Yaskawa INFORM job: DEMO_ROOF_SIDE_0625_3PAINT_6.JBI

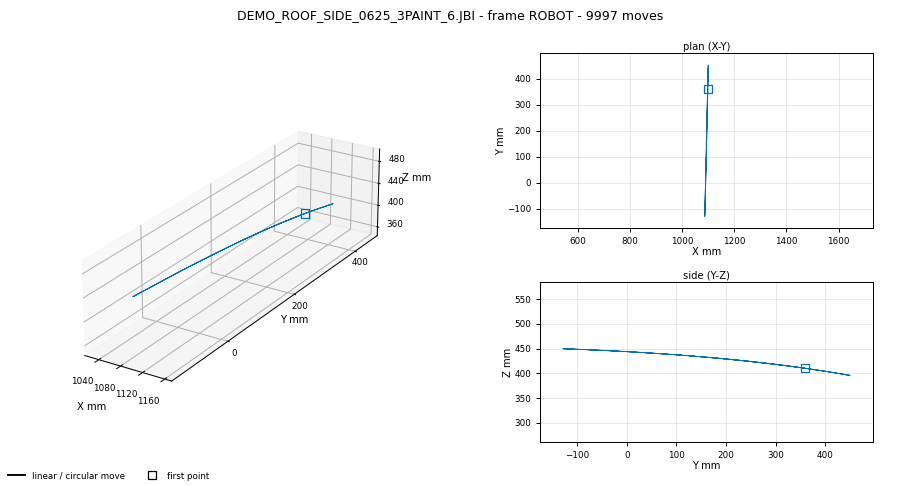
[picture p0: tool path of DEMO_ROOF_SIDE_0625_3PAINT_6.JBI in frame ROBOT, 9997 of 9997 moves have a stored position in this frame; points joined in program order, loops and branches not executed]
/JOB
//NAME DEMO_ROOF_SIDE_0625_3PAINT6
//POS
///NPOS 9997,0,0,0,0,0
///TOOL 0
///USER 0
///POSTYPE ROBOT
///RECTAN
///RCONF 1,0,0,0,0,0,0,0,0,0,0,0,0,0,0,0,0,0,0,0,0,0,0,0
C00000=1098.376,358.973,410.800,178.995,19.657,152.456
C00001=1098.369,358.726,410.835,178.993,19.653,152.456
C00002=1098.364,358.478,410.870,178.990,19.649,152.455
C00003=1098.358,358.230,410.905,178.986,19.645,152.455
C00004=1098.352,357.983,410.939,178.984,19.641,152.455
C00005=1098.347,357.735,410.974,178.980,19.637,152.454
C00006=1098.340,357.488,411.009,178.977,19.632,152.454
C00007=1098.332,357.110,411.062,178.973,19.626,152.453
C00008=1098.324,356.733,411.115,178.968,19.620,152.452
C00009=1098.314,356.355,411.168,178.964,19.614,152.452
C00010=1098.306,355.978,411.220,178.959,19.608,152.451
C00011=1098.300,355.731,411.256,178.956,19.604,152.451
C00012=1098.295,355.483,411.291,178.953,19.600,152.450
C00013=1098.289,355.235,411.325,178.950,19.596,152.450
C00014=1098.284,354.988,411.359,178.947,19.592,152.449
C00015=1098.277,354.740,411.395,178.944,19.588,152.449
C00016=1098.272,354.493,411.429,178.941,19.585,152.449
C00017=1098.266,354.245,411.463,178.938,19.580,152.448
C00018=1098.261,353.998,411.498,178.935,19.576,152.448
C00019=1098.254,353.750,411.532,178.932,19.572,152.447
C00020=1098.249,353.502,411.567,178.929,19.568,152.447
C00021=1098.243,353.255,411.601,178.926,19.565,152.446
C00022=1098.237,353.007,411.636,178.923,19.561,152.446
C00023=1098.231,352.760,411.671,178.919,19.557,152.446
C00024=1098.226,352.513,411.705,178.917,19.553,152.445
C00025=1098.220,352.265,411.740,178.913,19.549,152.445
C00026=1098.214,352.017,411.774,178.911,19.545,152.445
C00027=1098.208,351.770,411.808,178.907,19.541,152.444
C00028=1098.203,351.522,411.843,178.905,19.538,152.444
C00029=1098.197,351.275,411.877,178.901,19.534,152.443
C00030=1098.191,351.027,411.911,178.898,19.530,152.443
C00031=1098.186,350.779,411.945,178.895,19.526,152.443
C00032=1098.180,350.531,411.979,178.892,19.522,152.442
C00033=1098.174,350.284,412.013,178.889,19.519,152.442
C00034=1098.169,350.037,412.048,178.886,19.515,152.442
C00035=1098.163,349.789,412.082,178.883,19.512,152.441
C00036=1098.157,349.541,412.116,178.880,19.507,152.441
C00037=1098.151,349.294,412.150,178.877,19.504,152.441
C00038=1098.146,349.046,412.185,178.874,19.500,152.440
C00039=1098.140,348.799,412.218,178.871,19.497,152.440
C00040=1098.134,348.551,412.252,178.868,19.493,152.440
C00041=1098.128,348.303,412.287,178.865,19.489,152.439
C00042=1098.123,348.056,412.321,178.861,19.485,152.439
C00043=1098.117,347.808,412.355,178.859,19.482,152.439
C00044=1098.111,347.561,412.389,178.855,19.478,152.438
C00045=1098.105,347.313,412.423,178.853,19.475,152.438
C00046=1098.100,347.066,412.457,178.849,19.470,152.438
C00047=1098.095,346.818,412.491,178.847,19.467,152.437
C00048=1098.088,346.570,412.525,178.843,19.463,152.437
C00049=1098.082,346.322,412.559,178.840,19.460,152.437
C00050=1098.077,346.075,412.593,178.837,19.456,152.436
C00051=1098.071,345.827,412.627,178.834,19.453,152.436
C00052=1098.065,345.579,412.660,178.831,19.449,152.436
C00053=1098.060,345.332,412.695,178.828,19.445,152.435
C00054=1098.054,345.084,412.729,178.824,19.442,152.435
C00055=1098.049,344.837,412.762,178.822,19.438,152.435
C00056=1098.043,344.589,412.796,178.818,19.434,152.434
C00057=1098.038,344.341,412.830,178.815,19.431,152.434
C00058=1098.031,344.093,412.864,178.812,19.427,152.434
C00059=1098.022,343.718,412.915,178.808,19.422,152.433
C00060=1098.014,343.343,412.966,178.803,19.417,152.433
C00061=1098.005,342.968,413.017,178.798,19.412,152.433
C00062=1097.996,342.593,413.067,178.793,19.406,152.432
C00063=1097.990,342.345,413.101,178.790,19.403,152.432
C00064=1097.984,342.098,413.135,178.788,19.400,152.432
C00065=1097.979,341.850,413.169,178.784,19.396,152.431
C00066=1097.973,341.602,413.202,178.781,19.393,152.431
C00067=1097.967,341.354,413.236,178.778,19.389,152.431
C00068=1097.962,341.107,413.269,178.775,19.386,152.431
C00069=1097.956,340.859,413.303,178.771,19.382,152.430
C00070=1097.951,340.611,413.336,178.769,19.379,152.430
C00071=1097.945,340.363,413.370,178.766,19.376,152.430
C00072=1097.939,340.116,413.403,178.762,19.372,152.430
C00073=1097.934,339.868,413.437,178.759,19.369,152.429
C00074=1097.928,339.620,413.470,178.756,19.365,152.429
C00075=1097.922,339.373,413.503,178.753,19.362,152.429
C00076=1097.917,339.126,413.536,178.750,19.359,152.429
C00077=1097.911,338.878,413.570,178.747,19.355,152.428
C00078=1097.906,338.630,413.603,178.744,19.352,152.428
C00079=1097.900,338.382,413.636,178.740,19.349,152.428
C00080=1097.894,338.134,413.670,178.737,19.345,152.428
C00081=1097.888,337.887,413.703,178.735,19.342,152.427
C00082=1097.882,337.639,413.737,178.731,19.339,152.427
C00083=1097.877,337.391,413.770,178.728,19.335,152.427
C00084=1097.871,337.143,413.803,178.725,19.332,152.427
C00085=1097.865,336.896,413.836,178.722,19.329,152.427
C00086=1097.859,336.648,413.869,178.719,19.326,152.426
C00087=1097.854,336.400,413.903,178.715,19.322,152.426
C00088=1097.847,336.152,413.935,178.712,19.319,152.426
C00089=1097.842,335.904,413.969,178.709,19.316,152.426
C00090=1097.836,335.656,414.002,178.706,19.312,152.426
C00091=1097.831,335.409,414.035,178.703,19.309,152.425
C00092=1097.825,335.162,414.068,178.700,19.307,152.425
C00093=1097.820,334.914,414.101,178.696,19.303,152.425
C00094=1097.814,334.666,414.134,178.694,19.300,152.425
C00095=1097.808,334.418,414.167,178.691,19.297,152.424
C00096=1097.802,334.170,414.201,178.687,19.293,152.424
C00097=1097.797,333.922,414.233,178.684,19.290,152.424
C00098=1097.791,333.674,414.266,178.681,19.287,152.424
C00099=1097.786,333.427,414.299,178.678,19.283,152.424
C00100=1097.779,333.179,414.332,178.675,19.281,152.424
C00101=1097.774,332.932,414.365,178.672,19.278,152.423
C00102=1097.769,332.683,414.398,178.668,19.274,152.423
C00103=1097.762,332.435,414.430,178.665,19.271,152.423
C00104=1097.757,332.187,414.464,178.662,19.268,152.423
C00105=1097.751,331.941,414.496,178.659,19.265,152.423
C00106=1097.745,331.693,414.529,178.656,19.262,152.423
C00107=1097.739,331.444,414.561,178.653,19.259,152.422
C00108=1097.734,331.197,414.595,178.650,19.256,152.422
C00109=1097.728,330.949,414.627,178.646,19.253,152.422
C00110=1097.722,330.701,414.660,178.643,19.250,152.422
C00111=1097.713,330.320,414.710,178.638,19.245,152.422
C00112=1097.704,329.938,414.760,178.634,19.240,152.421
C00113=1097.695,329.558,414.811,178.628,19.236,152.421
C00114=1097.686,329.176,414.861,178.624,19.231,152.421
C00115=1097.680,328.929,414.893,178.620,19.228,152.421
C00116=1097.675,328.680,414.926,178.617,19.225,152.421
C00117=1097.669,328.432,414.959,178.614,19.222,152.421
C00118=1097.663,328.185,414.990,178.611,19.220,152.421
C00119=1097.658,327.937,415.024,178.607,19.216,152.420
C00120=1097.652,327.689,415.056,178.605,19.213,152.420
C00121=1097.645,327.441,415.088,178.602,19.211,152.420
C00122=1097.640,327.194,415.120,178.598,19.208,152.420
C00123=1097.634,326.946,415.153,178.595,19.204,152.420
C00124=1097.628,326.698,415.186,178.592,19.201,152.420
C00125=1097.622,326.450,415.218,178.589,19.199,152.420
C00126=1097.618,326.202,415.251,178.586,19.196,152.420
C00127=1097.612,325.954,415.283,178.582,19.193,152.420
C00128=1097.605,325.706,415.315,178.579,19.190,152.419
C00129=1097.600,325.459,415.347,178.576,19.187,152.419
C00130=1097.595,325.210,415.380,178.573,19.184,152.419
C00131=1097.588,324.963,415.412,178.569,19.181,152.419
C00132=1097.583,324.715,415.444,178.566,19.178,152.419
C00133=1097.577,324.467,415.476,178.563,19.175,152.419
C00134=1097.571,324.219,415.509,178.560,19.173,152.419
C00135=1097.566,323.972,415.541,178.557,19.170,152.419
C00136=1097.560,323.723,415.573,178.553,19.167,152.418
C00137=1097.554,323.475,415.605,178.550,19.164,152.418
C00138=1097.548,323.228,415.637,178.547,19.161,152.418
C00139=1097.543,322.980,415.670,178.544,19.158,152.418
C00140=1097.538,322.732,415.702,178.542,19.155,152.418
C00141=1097.532,322.484,415.734,178.538,19.152,152.418
C00142=1097.526,322.236,415.766,178.535,19.149,152.418
C00143=1097.520,321.989,415.798,178.532,19.147,152.418
C00144=1097.514,321.741,415.830,178.529,19.144,152.418
C00145=1097.509,321.493,415.862,178.526,19.141,152.418
C00146=1097.503,321.245,415.894,178.522,19.138,152.417
C00147=1097.497,320.996,415.926,178.519,19.135,152.417
C00148=1097.492,320.749,415.958,178.516,19.133,152.417
C00149=1097.486,320.501,415.990,178.513,19.130,152.417
C00150=1097.481,320.253,416.022,178.510,19.127,152.417
C00151=1097.475,320.005,416.054,178.507,19.125,152.417
C00152=1097.469,319.757,416.086,178.503,19.121,152.417
C00153=1097.464,319.509,416.118,178.500,19.119,152.417
C00154=1097.459,319.261,416.150,178.497,19.116,152.417
C00155=1097.453,319.013,416.182,178.494,19.113,152.417
C00156=1097.447,318.766,416.213,178.491,19.111,152.417
C00157=1097.441,318.517,416.246,178.488,19.108,152.417
C00158=1097.436,318.270,416.277,178.484,19.105,152.416
C00159=1097.430,318.022,416.309,178.481,19.102,152.416
C00160=1097.425,317.774,416.341,178.478,19.099,152.416
C00161=1097.419,317.527,416.373,178.475,19.097,152.416
C00162=1097.413,317.279,416.405,178.472,19.094,152.416
C00163=1097.405,316.890,416.454,178.466,19.089,152.416
C00164=1097.397,316.502,416.504,178.462,19.085,152.416
C00165=1097.387,316.114,416.553,178.456,19.081,152.416
C00166=1097.379,315.725,416.603,178.452,19.077,152.416
C00167=1097.373,315.478,416.635,178.449,19.074,152.416
C00168=1097.368,315.229,416.666,178.445,19.071,152.416
C00169=1097.362,314.981,416.698,178.442,19.068,152.416
C00170=1097.356,314.734,416.729,178.439,19.066,152.416
C00171=1097.350,314.486,416.761,178.435,19.063,152.416
C00172=1097.344,314.237,416.792,178.432,19.061,152.416
C00173=1097.338,313.990,416.823,178.429,19.058,152.416
C00174=1097.332,313.742,416.855,178.426,19.056,152.415
C00175=1097.327,313.494,416.886,178.423,19.053,152.416
C00176=1097.321,313.246,416.918,178.420,19.051,152.415
C00177=1097.315,312.998,416.949,178.416,19.047,152.415
C00178=1097.310,312.750,416.980,178.412,19.045,152.415
C00179=1097.303,312.502,417.012,178.409,19.043,152.415
C00180=1097.298,312.255,417.043,178.406,19.040,152.415
C00181=1097.292,312.006,417.075,178.403,19.038,152.415
C00182=1097.286,311.759,417.106,178.400,19.035,152.415
C00183=1097.280,311.510,417.137,178.397,19.033,152.415
C00184=1097.275,311.262,417.169,178.394,19.030,152.415
C00185=1097.269,311.014,417.199,178.391,19.028,152.415
C00186=1097.263,310.766,417.231,178.387,19.025,152.415
C00187=1097.257,310.518,417.261,178.384,19.023,152.415
C00188=1097.252,310.271,417.293,178.380,19.020,152.415
C00189=1097.246,310.022,417.324,178.377,19.017,152.415
C00190=1097.240,309.775,417.355,178.374,19.015,152.415
C00191=1097.235,309.527,417.386,178.371,19.013,152.415
C00192=1097.228,309.279,417.418,178.367,19.010,152.415
C00193=1097.223,309.031,417.449,178.364,19.008,152.415
C00194=1097.217,308.783,417.480,178.361,19.005,152.415
C00195=1097.212,308.535,417.511,178.358,19.003,152.415
C00196=1097.207,308.287,417.542,178.355,19.000,152.415
C00197=1097.200,308.039,417.573,178.352,18.998,152.415
C00198=1097.195,307.791,417.604,178.348,18.996,152.416
C00199=1097.189,307.543,417.635,178.345,18.993,152.415
C00200=1097.183,307.295,417.666,178.342,18.991,152.415
C00201=1097.178,307.047,417.697,178.339,18.988,152.415
C00202=1097.173,306.799,417.728,178.335,18.985,152.416
C00203=1097.166,306.551,417.758,178.332,18.983,152.416
C00204=1097.161,306.303,417.790,178.329,18.980,152.415
C00205=1097.155,306.055,417.820,178.325,18.978,152.416
C00206=1097.150,305.807,417.851,178.322,18.975,152.415
C00207=1097.143,305.559,417.882,178.319,18.973,152.416
C00208=1097.138,305.311,417.914,178.316,18.971,152.416
C00209=1097.132,305.063,417.944,178.313,18.968,152.416
C00210=1097.127,304.815,417.975,178.309,18.966,152.416
C00211=1097.121,304.567,418.005,178.306,18.963,152.416
C00212=1097.116,304.320,418.036,178.303,18.961,152.416
C00213=1097.110,304.071,418.067,178.300,18.958,152.416
C00214=1097.104,303.824,418.098,178.297,18.956,152.416
C00215=1097.096,303.437,418.145,178.291,18.952,152.416
C00216=1097.087,303.052,418.193,178.286,18.948,152.416
C00217=1097.077,302.666,418.241,178.281,18.945,152.416
C00218=1097.069,302.281,418.289,178.277,18.941,152.416
C00219=1097.064,302.032,418.320,178.273,18.939,152.416
C00220=1097.058,301.785,418.350,178.270,18.936,152.416
C00221=1097.052,301.537,418.381,178.267,18.934,152.416
C00222=1097.047,301.289,418.412,178.264,18.932,152.416
C00223=1097.041,301.041,418.442,178.260,18.928,152.416
C00224=1097.036,300.793,418.472,178.257,18.926,152.416
C00225=1097.031,300.545,418.503,178.253,18.924,152.416
C00226=1097.025,300.296,418.533,178.250,18.922,152.416
C00227=1097.019,300.049,418.563,178.247,18.919,152.416
C00228=1097.014,299.801,418.594,178.244,18.917,152.416
C00229=1097.008,299.553,418.624,178.240,18.914,152.416
C00230=1097.002,299.305,418.655,178.237,18.912,152.416
C00231=1096.997,299.057,418.686,178.234,18.910,152.416
C00232=1096.992,298.809,418.716,178.231,18.907,152.416
C00233=1096.986,298.560,418.746,178.228,18.905,152.416
C00234=1096.981,298.312,418.777,178.224,18.903,152.416
C00235=1096.975,298.065,418.807,178.221,18.900,152.417
C00236=1096.969,297.816,418.838,178.218,18.898,152.417
C00237=1096.963,297.568,418.867,178.214,18.896,152.417
C00238=1096.957,297.320,418.898,178.211,18.894,152.417
C00239=1096.952,297.072,418.928,178.208,18.891,152.417
C00240=1096.947,296.824,418.959,178.205,18.889,152.417
C00241=1096.941,296.575,418.989,178.202,18.887,152.417
C00242=1096.935,296.328,419.019,178.199,18.885,152.417
C00243=1096.929,296.080,419.049,178.196,18.883,152.417
C00244=1096.924,295.831,419.079,178.193,18.880,152.417
C00245=1096.918,295.583,419.109,178.189,18.878,152.417
C00246=1096.912,295.336,419.140,178.186,18.876,152.417
C00247=1096.907,295.087,419.169,178.183,18.874,152.417
C00248=1096.901,294.839,419.200,178.179,18.871,152.417
C00249=1096.895,294.591,419.229,178.176,18.869,152.418
C00250=1096.890,294.343,419.260,178.173,18.867,152.418
C00251=1096.884,294.095,419.289,178.169,18.865,152.418
C00252=1096.878,293.847,419.320,178.166,18.863,152.418
C00253=1096.872,293.599,419.350,178.163,18.860,152.418
C00254=1096.867,293.351,419.380,178.160,18.858,152.418
C00255=1096.861,293.103,419.410,178.156,18.856,152.418
C00256=1096.856,292.854,419.440,178.153,18.854,152.418
C00257=1096.850,292.606,419.469,178.150,18.851,152.418
C00258=1096.844,292.358,419.500,178.146,18.849,152.418
C00259=1096.839,292.110,419.529,178.143,18.847,152.418
C00260=1096.833,291.862,419.560,178.140,18.845,152.418
C00261=1096.828,291.614,419.589,178.137,18.842,152.419
C00262=1096.822,291.366,419.619,178.134,18.841,152.419
C00263=1096.816,291.118,419.648,178.131,18.839,152.419
C00264=1096.810,290.870,419.678,178.127,18.837,152.419
C00265=1096.805,290.622,419.708,178.124,18.834,152.419
C00266=1096.799,290.373,419.738,178.121,18.832,152.419
C00267=1096.791,290.001,419.783,178.116,18.829,152.419
C00268=1096.782,289.630,419.827,178.111,18.826,152.419
C00269=1096.774,289.258,419.872,178.106,18.822,152.420
C00270=1096.765,288.887,419.916,178.101,18.819,152.420
C00271=1096.759,288.638,419.946,178.098,18.817,152.420
C00272=1096.754,288.390,419.975,178.095,18.815,152.420
C00273=1096.748,288.141,420.005,178.092,18.813,152.420
C00274=1096.742,287.894,420.035,178.088,18.811,152.420
C00275=1096.736,287.645,420.064,178.085,18.809,152.420
C00276=1096.731,287.398,420.094,178.082,18.807,152.420
C00277=1096.726,287.149,420.123,178.078,18.805,152.420
C00278=1096.720,286.901,420.152,178.075,18.802,152.421
C00279=1096.714,286.653,420.182,178.071,18.801,152.421
C00280=1096.709,286.404,420.211,178.068,18.798,152.421
C00281=1096.702,286.157,420.241,178.066,18.797,152.421
C00282=1096.697,285.909,420.270,178.062,18.794,152.421
C00283=1096.692,285.660,420.300,178.059,18.793,152.421
C00284=1096.685,285.412,420.329,178.056,18.790,152.421
C00285=1096.680,285.164,420.359,178.052,18.788,152.421
C00286=1096.674,284.915,420.388,178.049,18.786,152.422
C00287=1096.669,284.668,420.417,178.046,18.784,152.422
C00288=1096.663,284.420,420.447,178.042,18.782,152.422
C00289=1096.658,284.171,420.476,178.040,18.780,152.422
C00290=1096.651,283.923,420.505,178.036,18.778,152.422
C00291=1096.646,283.675,420.535,178.033,18.776,152.422
C00292=1096.641,283.427,420.564,178.030,18.774,152.422
C00293=1096.635,283.179,420.593,178.026,18.772,152.422
C00294=1096.629,282.930,420.623,178.023,18.770,152.423
C00295=1096.624,282.681,420.652,178.020,18.767,152.423
C00296=1096.618,282.434,420.681,178.016,18.766,152.423
C00297=1096.613,282.185,420.710,178.014,18.764,152.423
C00298=1096.607,281.937,420.739,178.010,18.762,152.423
C00299=1096.602,281.689,420.769,178.007,18.760,152.423
C00300=1096.595,281.441,420.798,178.004,18.758,152.423
C00301=1096.590,281.193,420.827,178.000,18.755,152.423
C00302=1096.584,280.944,420.856,177.997,18.754,152.424
C00303=1096.579,280.696,420.885,177.994,18.751,152.424
C00304=1096.573,280.448,420.914,177.991,18.750,152.424
C00305=1096.567,280.200,420.943,177.988,18.748,152.424
C00306=1096.561,279.951,420.972,177.984,18.746,152.424
C00307=1096.556,279.703,421.001,177.981,18.744,152.424
C00308=1096.550,279.455,421.030,177.977,18.741,152.424
C00309=1096.545,279.207,421.060,177.974,18.740,152.425
C00310=1096.539,278.959,421.088,177.971,18.738,152.425
C00311=1096.533,278.711,421.117,177.968,18.736,152.425
C00312=1096.528,278.462,421.146,177.965,18.734,152.425
C00313=1096.522,278.214,421.174,177.961,18.732,152.425
C00314=1096.517,277.966,421.204,177.958,18.730,152.425
C00315=1096.511,277.717,421.232,177.954,18.728,152.426
C00316=1096.505,277.469,421.261,177.952,18.726,152.426
C00317=1096.500,277.221,421.291,177.948,18.724,152.426
C00318=1096.494,276.972,421.319,177.945,18.722,152.426
C00319=1096.486,276.610,421.361,177.940,18.719,152.426
C00320=1096.478,276.248,421.403,177.936,18.717,152.427
C00321=1096.469,275.885,421.445,177.931,18.714,152.427
C00322=1096.460,275.523,421.487,177.926,18.711,152.427
C00323=1096.456,275.275,421.515,177.923,18.709,152.427
C00324=1096.450,275.026,421.545,177.920,18.707,152.427
C00325=1096.444,274.778,421.573,177.916,18.705,152.427
C00326=1096.439,274.530,421.602,177.913,18.703,152.428
C00327=1096.433,274.281,421.630,177.910,18.702,152.428
C00328=1096.427,274.034,421.659,177.907,18.700,152.428
C00329=1096.421,273.785,421.687,177.903,18.698,152.428
C00330=1096.416,273.536,421.716,177.900,18.696,152.428
C00331=1096.410,273.289,421.745,177.896,18.694,152.428
C00332=1096.404,273.040,421.773,177.894,18.692,152.429
C00333=1096.399,272.792,421.802,177.890,18.690,152.429
C00334=1096.393,272.544,421.830,177.887,18.688,152.429
C00335=1096.388,272.295,421.859,177.884,18.686,152.429
C00336=1096.382,272.046,421.887,177.881,18.685,152.429
C00337=1096.376,271.798,421.916,177.877,18.683,152.430
C00338=1096.371,271.550,421.944,177.874,18.681,152.430
C00339=1096.365,271.302,421.973,177.871,18.679,152.430
C00340=1096.359,271.054,422.001,177.867,18.677,152.430
C00341=1096.353,270.805,422.030,177.865,18.676,152.430
C00342=1096.349,270.557,422.058,177.861,18.674,152.430
C00343=1096.343,270.308,422.086,177.858,18.671,152.430
C00344=1096.337,270.060,422.114,177.854,18.670,152.431
C00345=1096.331,269.812,422.143,177.852,18.668,152.431
C00346=1096.326,269.564,422.171,177.848,18.666,152.431
C00347=1096.320,269.315,422.200,177.845,18.664,152.431
C00348=1096.314,269.067,422.228,177.841,18.663,152.431
C00349=1096.308,268.818,422.256,177.838,18.660,152.432
C00350=1096.303,268.570,422.284,177.835,18.659,152.432
C00351=1096.297,268.322,422.312,177.832,18.657,152.432
C00352=1096.292,268.074,422.341,177.828,18.655,152.432
C00353=1096.286,267.825,422.369,177.825,18.653,152.432
C00354=1096.280,267.577,422.397,177.822,18.652,152.433
C00355=1096.274,267.329,422.426,177.819,18.650,152.433
C00356=1096.269,267.081,422.454,177.815,18.648,152.433
C00357=1096.263,266.832,422.482,177.812,18.646,152.433
C00358=1096.258,266.584,422.510,177.809,18.644,152.433
C00359=1096.252,266.335,422.538,177.806,18.643,152.433
C00360=1096.246,266.087,422.566,177.802,18.641,152.434
C00361=1096.241,265.839,422.594,177.799,18.639,152.434
C00362=1096.235,265.590,422.622,177.796,18.637,152.434
C00363=1096.230,265.342,422.650,177.793,18.636,152.434
C00364=1096.224,265.093,422.678,177.789,18.634,152.434
C00365=1096.219,264.845,422.706,177.786,18.631,152.435
C00366=1096.213,264.597,422.734,177.783,18.630,152.435
C00367=1096.207,264.348,422.762,177.780,18.628,152.435
C00368=1096.201,264.100,422.790,177.776,18.627,152.435
C00369=1096.195,263.851,422.818,177.773,18.625,152.435
C00370=1096.190,263.603,422.846,177.770,18.623,152.436
C00371=1096.182,263.243,422.885,177.765,18.621,152.436
C00372=1096.173,262.884,422.926,177.760,18.618,152.436
C00373=1096.165,262.525,422.966,177.756,18.616,152.437
C00374=1096.157,262.164,423.006,177.751,18.613,152.437
C00375=1096.151,261.916,423.034,177.748,18.612,152.437
C00376=1096.145,261.668,423.062,177.745,18.610,152.437
C00377=1096.139,261.420,423.090,177.741,18.608,152.438
C00378=1096.134,261.171,423.117,177.738,18.606,152.438
C00379=1096.128,260.923,423.145,177.735,18.605,152.438
C00380=1096.122,260.674,423.173,177.731,18.603,152.438
C00381=1096.116,260.426,423.201,177.728,18.602,152.439
C00382=1096.111,260.178,423.228,177.725,18.600,152.439
C00383=1096.105,259.929,423.256,177.722,18.598,152.439
C00384=1096.100,259.680,423.283,177.718,18.596,152.439
C00385=1096.094,259.432,423.311,177.716,18.595,152.439
C00386=1096.088,259.184,423.339,177.712,18.593,152.440
C00387=1096.083,258.935,423.366,177.709,18.591,152.440
C00388=1096.076,258.687,423.394,177.705,18.590,152.440
C00389=1096.071,258.438,423.421,177.702,18.588,152.440
C00390=1096.065,258.190,423.449,177.699,18.586,152.440
C00391=1096.060,257.942,423.476,177.695,18.584,152.441
C00392=1096.054,257.693,423.504,177.693,18.583,152.441
C00393=1096.048,257.445,423.531,177.689,18.581,152.441
C00394=1096.043,257.196,423.559,177.686,18.580,152.441
C00395=1096.037,256.948,423.585,177.683,18.578,152.442
C00396=1096.031,256.699,423.614,177.679,18.576,152.442
C00397=1096.026,256.451,423.641,177.676,18.575,152.442
C00398=1096.020,256.203,423.668,177.673,18.573,152.442
C00399=1096.015,255.954,423.695,177.670,18.571,152.442
C00400=1096.008,255.706,423.723,177.666,18.569,152.443
C00401=1096.003,255.457,423.750,177.664,18.568,152.443
C00402=1095.997,255.209,423.777,177.660,18.566,152.443
C00403=1095.992,254.961,423.805,177.657,18.565,152.443
C00404=1095.986,254.712,423.832,177.654,18.563,152.444
C00405=1095.980,254.464,423.860,177.650,18.562,152.444
C00406=1095.974,254.215,423.887,177.647,18.560,152.444
C00407=1095.969,253.966,423.914,177.644,18.558,152.444
C00408=1095.963,253.719,423.941,177.641,18.556,152.444
C00409=1095.958,253.469,423.969,177.637,18.554,152.445
C00410=1095.952,253.221,423.996,177.635,18.553,152.445
C00411=1095.947,252.972,424.023,177.631,18.551,152.445
C00412=1095.941,252.725,424.050,177.628,18.550,152.445
C00413=1095.936,252.476,424.077,177.625,18.548,152.446
C00414=1095.930,252.228,424.104,177.621,18.547,152.446
C00415=1095.924,251.978,424.132,177.618,18.544,152.446
C00416=1095.919,251.730,424.158,177.615,18.543,152.446
C00417=1095.913,251.482,424.186,177.612,18.541,152.446
C00418=1095.908,251.233,424.213,177.608,18.540,152.447
C00419=1095.902,250.985,424.240,177.606,18.538,152.447
C00420=1095.897,250.736,424.267,177.602,18.536,152.447
C00421=1095.892,250.488,424.294,177.598,18.535,152.447
C00422=1095.886,250.239,424.321,177.596,18.533,152.448
C00423=1095.877,249.877,424.361,177.591,18.531,152.448
C00424=1095.869,249.514,424.400,177.586,18.528,152.448
C00425=1095.862,249.152,424.439,177.582,18.526,152.448
C00426=1095.853,248.789,424.479,177.576,18.523,152.449
C00427=1095.847,248.540,424.506,177.574,18.522,152.449
C00428=1095.842,248.292,424.532,177.570,18.520,152.449
C00429=1095.837,248.043,424.559,177.567,18.518,152.449
C00430=1095.831,247.795,424.586,177.564,18.517,152.450
C00431=1095.826,247.546,424.613,177.561,18.515,152.450
C00432=1095.820,247.298,424.640,177.558,18.514,152.450
C00433=1095.814,247.050,424.667,177.554,18.512,152.450
C00434=1095.809,246.801,424.693,177.551,18.510,152.451
C00435=1095.804,246.553,424.721,177.548,18.509,152.451
C00436=1095.798,246.304,424.747,177.545,18.507,152.451
C00437=1095.792,246.055,424.773,177.541,18.505,152.451
C00438=1095.786,245.807,424.800,177.538,18.504,152.452
C00439=1095.781,245.559,424.826,177.535,18.502,152.452
C00440=1095.776,245.310,424.854,177.532,18.501,152.452
C00441=1095.770,245.062,424.880,177.529,18.499,152.452
C00442=1095.764,244.813,424.907,177.525,18.498,152.453
C00443=1095.758,244.565,424.934,177.522,18.496,152.453
C00444=1095.753,244.316,424.960,177.519,18.495,152.453
C00445=1095.748,244.067,424.987,177.516,18.493,152.453
C00446=1095.742,243.819,425.013,177.513,18.492,152.454
C00447=1095.736,243.570,425.040,177.509,18.490,152.454
C00448=1095.731,243.321,425.066,177.506,18.489,152.454
C00449=1095.725,243.073,425.093,177.503,18.487,152.454
C00450=1095.719,242.825,425.119,177.500,18.486,152.454
C00451=1095.714,242.576,425.146,177.497,18.484,152.455
C00452=1095.708,242.327,425.172,177.493,18.482,152.455
C00453=1095.702,242.079,425.199,177.490,18.481,152.455
C00454=1095.697,241.831,425.225,177.487,18.479,152.455
C00455=1095.691,241.582,425.251,177.484,18.478,152.456
C00456=1095.685,241.333,425.278,177.481,18.476,152.456
C00457=1095.679,241.085,425.304,177.478,18.475,152.456
C00458=1095.674,240.836,425.330,177.474,18.473,152.456
C00459=1095.668,240.588,425.357,177.471,18.471,152.457
C00460=1095.663,240.339,425.383,177.468,18.470,152.457
C00461=1095.657,240.090,425.410,177.465,18.468,152.457
C00462=1095.651,239.842,425.436,177.462,18.467,152.457
C00463=1095.646,239.593,425.462,177.458,18.466,152.458
C00464=1095.640,239.345,425.489,177.454,18.464,152.458
C00465=1095.635,239.096,425.515,177.452,18.462,152.458
C00466=1095.629,238.847,425.541,177.448,18.461,152.459
C00467=1095.623,238.598,425.567,177.446,18.459,152.459
C00468=1095.618,238.350,425.594,177.442,18.458,152.459
C00469=1095.613,238.102,425.620,177.439,18.456,152.459
C00470=1095.607,237.853,425.646,177.436,18.455,152.460
C00471=1095.601,237.604,425.672,177.433,18.453,152.460
C00472=1095.595,237.356,425.698,177.429,18.452,152.460
C00473=1095.589,237.107,425.724,177.426,18.450,152.460
C00474=1095.584,236.858,425.750,177.423,18.449,152.460
C00475=1095.576,236.489,425.789,177.419,18.447,152.461
C00476=1095.567,236.120,425.827,177.413,18.444,152.461
C00477=1095.559,235.751,425.867,177.409,18.442,152.462
C00478=1095.551,235.381,425.905,177.404,18.440,152.462
C00479=1095.545,235.133,425.931,177.401,18.438,152.462
C00480=1095.540,234.884,425.957,177.398,18.437,152.463
C00481=1095.534,234.635,425.983,177.394,18.435,152.463
C00482=1095.529,234.386,426.009,177.392,18.434,152.463
C00483=1095.523,234.138,426.035,177.388,18.432,152.463
C00484=1095.517,233.889,426.061,177.385,18.431,152.464
C00485=1095.512,233.640,426.087,177.382,18.429,152.464
C00486=1095.506,233.392,426.113,177.378,18.427,152.464
C00487=1095.500,233.143,426.139,177.375,18.427,152.464
C00488=1095.495,232.895,426.164,177.372,18.425,152.465
C00489=1095.489,232.646,426.190,177.369,18.424,152.465
C00490=1095.484,232.397,426.216,177.366,18.422,152.465
C00491=1095.478,232.149,426.242,177.363,18.421,152.465
C00492=1095.472,231.900,426.268,177.359,18.419,152.466
C00493=1095.467,231.652,426.294,177.357,18.418,152.466
C00494=1095.461,231.403,426.319,177.353,18.416,152.466
C00495=1095.456,231.154,426.345,177.350,18.415,152.466
C00496=1095.450,230.905,426.371,177.347,18.413,152.467
C00497=1095.445,230.657,426.397,177.344,18.412,152.467
C00498=1095.439,230.408,426.422,177.340,18.410,152.467
C00499=1095.433,230.159,426.448,177.338,18.409,152.468
C00500=1095.427,229.911,426.474,177.334,18.407,152.468
C00501=1095.422,229.663,426.499,177.331,18.406,152.468
C00502=1095.416,229.414,426.525,177.328,18.404,152.468
C00503=1095.410,229.165,426.551,177.325,18.404,152.469
C00504=1095.404,228.917,426.576,177.321,18.402,152.469
C00505=1095.399,228.668,426.602,177.319,18.401,152.469
C00506=1095.394,228.419,426.628,177.315,18.399,152.469
C00507=1095.388,228.171,426.653,177.312,18.398,152.470
C00508=1095.382,227.922,426.679,177.309,18.396,152.470
C00509=1095.377,227.674,426.704,177.306,18.395,152.470
C00510=1095.371,227.425,426.730,177.302,18.393,152.471
C00511=1095.365,227.176,426.754,177.300,18.392,152.471
C00512=1095.360,226.927,426.780,177.296,18.390,152.471
C00513=1095.354,226.679,426.805,177.293,18.389,152.471
C00514=1095.349,226.430,426.831,177.290,18.387,152.472
C00515=1095.343,226.182,426.856,177.287,18.386,152.472
C00516=1095.337,225.933,426.881,177.283,18.385,152.472
C00517=1095.331,225.684,426.907,177.281,18.383,152.472
C00518=1095.326,225.436,426.932,177.277,18.382,152.473
C00519=1095.321,225.186,426.958,177.274,18.380,152.473
C00520=1095.314,224.938,426.983,177.271,18.379,152.473
C00521=1095.310,224.689,427.009,177.268,18.378,152.474
C00522=1095.303,224.441,427.034,177.264,18.376,152.474
C00523=1095.298,224.192,427.060,177.262,18.375,152.474
C00524=1095.293,223.943,427.084,177.258,18.373,152.474
C00525=1095.286,223.695,427.109,177.255,18.372,152.475
C00526=1095.282,223.446,427.135,177.252,18.370,152.475
C00527=1095.273,223.068,427.174,177.247,18.368,152.475
C00528=1095.265,222.689,427.211,177.243,18.366,152.476
C00529=1095.256,222.312,427.250,177.238,18.364,152.476
C00530=1095.247,221.934,427.288,177.233,18.362,152.477
C00531=1095.242,221.685,427.314,177.230,18.360,152.477
C00532=1095.236,221.436,427.338,177.227,18.360,152.477
C00533=1095.230,221.188,427.363,177.224,18.358,152.477
C00534=1095.225,220.940,427.388,177.221,18.357,152.478
C00535=1095.219,220.690,427.414,177.217,18.355,152.478
C00536=1095.213,220.442,427.439,177.214,18.354,152.478
C00537=1095.208,220.193,427.463,177.211,18.352,152.479
C00538=1095.202,219.944,427.488,177.208,18.351,152.479
C00539=1095.197,219.695,427.513,177.205,18.349,152.479
C00540=1095.191,219.447,427.539,177.202,18.348,152.479
C00541=1095.186,219.198,427.563,177.198,18.347,152.480
C00542=1095.179,218.949,427.588,177.195,18.345,152.480
C00543=1095.174,218.701,427.612,177.193,18.344,152.480
C00544=1095.169,218.452,427.638,177.189,18.342,152.480
C00545=1095.163,218.203,427.663,177.186,18.342,152.481
C00546=1095.157,217.955,427.688,177.183,18.340,152.481
C00547=1095.151,217.705,427.713,177.180,18.339,152.481
C00548=1095.146,217.457,427.738,177.176,18.337,152.482
C00549=1095.140,217.208,427.762,177.174,18.336,152.482
C00550=1095.135,216.960,427.788,177.171,18.335,152.482
C00551=1095.130,216.711,427.812,177.167,18.333,152.483
C00552=1095.124,216.462,427.837,177.164,18.332,152.483
C00553=1095.118,216.214,427.862,177.161,18.330,152.483
C00554=1095.112,215.965,427.886,177.158,18.329,152.483
C00555=1095.107,215.717,427.911,177.154,18.328,152.484
C00556=1095.101,215.467,427.936,177.152,18.326,152.484
C00557=1095.095,215.219,427.960,177.149,18.325,152.484
C00558=1095.090,214.970,427.986,177.145,18.323,152.484
C00559=1095.085,214.721,428.010,177.143,18.322,152.485
C00560=1095.079,214.473,428.035,177.139,18.321,152.485
C00561=1095.073,214.223,428.059,177.136,18.320,152.485
C00562=1095.068,213.975,428.084,177.133,18.319,152.486
C00563=1095.062,213.726,428.109,177.130,18.317,152.486
C00564=1095.057,213.478,428.133,177.127,18.316,152.486
C00565=1095.051,213.229,428.157,177.124,18.314,152.486
C00566=1095.045,212.980,428.183,177.121,18.313,152.487
C00567=1095.040,212.732,428.207,177.118,18.312,152.487
C00568=1095.034,212.482,428.232,177.114,18.310,152.487
C00569=1095.029,212.234,428.256,177.112,18.309,152.487
C00570=1095.023,211.985,428.280,177.108,18.307,152.488
C00571=1095.017,211.737,428.305,177.105,18.306,152.488
C00572=1095.012,211.488,428.330,177.102,18.305,152.488
C00573=1095.006,211.239,428.354,177.099,18.303,152.489
C00574=1095.001,210.990,428.378,177.096,18.302,152.489
C00575=1094.995,210.742,428.403,177.092,18.301,152.489
C00576=1094.989,210.492,428.427,177.090,18.300,152.490
C00577=1094.984,210.244,428.452,177.087,18.298,152.490
C00578=1094.978,209.995,428.475,177.083,18.297,152.490
C00579=1094.970,209.621,428.512,177.079,18.295,152.490
C00580=1094.961,209.247,428.549,177.074,18.293,152.491
C00581=1094.952,208.872,428.585,177.070,18.291,152.491
C00582=1094.944,208.498,428.622,177.065,18.289,152.492
C00583=1094.921,207.483,428.720,177.011,18.266,152.497
C00584=1094.916,207.234,428.744,177.008,18.266,152.497
C00585=1094.910,206.986,428.768,177.005,18.265,152.498
C00586=1094.904,206.737,428.793,177.002,18.265,152.498
C00587=1094.899,206.488,428.816,176.998,18.264,152.499
C00588=1094.893,206.239,428.840,176.995,18.264,152.499
C00589=1094.888,205.991,428.864,176.991,18.263,152.500
C00590=1094.882,205.741,428.889,176.988,18.262,152.500
C00591=1094.876,205.492,428.912,176.985,18.262,152.501
C00592=1094.871,205.244,428.936,176.982,18.262,152.501
C00593=1094.865,204.996,428.960,176.979,18.261,152.502
C00594=1094.860,204.746,428.983,176.975,18.261,152.502
C00595=1094.855,204.498,429.007,176.972,18.261,152.503
C00596=1094.848,204.249,429.031,176.969,18.260,152.503
C00597=1094.843,204.000,429.055,176.966,18.260,152.504
C00598=1094.837,203.751,429.079,176.963,18.259,152.504
C00599=1094.832,203.503,429.103,176.960,18.259,152.505
C00600=1094.827,203.254,429.126,176.956,18.258,152.505
C00601=1094.821,203.005,429.150,176.953,18.258,152.506
C00602=1094.816,202.756,429.174,176.949,18.257,152.506
C00603=1094.809,202.507,429.198,176.946,18.256,152.507
C00604=1094.804,202.258,429.221,176.943,18.256,152.507
C00605=1094.798,202.010,429.245,176.940,18.256,152.508
C00606=1094.792,201.761,429.268,176.937,18.255,152.508
C00607=1094.787,201.512,429.292,176.933,18.255,152.509
C00608=1094.780,201.263,429.316,176.930,18.255,152.509
C00609=1094.775,201.014,429.340,176.927,18.254,152.510
C00610=1094.769,200.766,429.363,176.924,18.254,152.510
C00611=1094.764,200.517,429.386,176.921,18.253,152.511
C00612=1094.758,200.268,429.410,176.917,18.253,152.511
C00613=1094.752,200.019,429.433,176.914,18.253,152.512
C00614=1094.747,199.770,429.456,176.911,18.252,152.512
C00615=1094.741,199.521,429.481,176.908,18.252,152.513
C00616=1094.735,199.272,429.504,176.905,18.251,152.514
C00617=1094.729,199.024,429.528,176.902,18.251,152.514
C00618=1094.724,198.775,429.551,176.898,18.250,152.514
C00619=1094.718,198.526,429.574,176.895,18.250,152.515
C00620=1094.712,198.278,429.598,176.892,18.249,152.515
C00621=1094.707,198.028,429.621,176.889,18.249,152.516
C00622=1094.701,197.780,429.645,176.886,18.249,152.517
C00623=1094.696,197.531,429.668,176.882,18.248,152.517
C00624=1094.691,197.282,429.691,176.879,18.247,152.517
C00625=1094.685,197.034,429.715,176.875,18.247,152.518
C00626=1094.678,196.784,429.738,176.872,18.246,152.518
C00627=1094.673,196.535,429.762,176.869,18.246,152.519
C00628=1094.667,196.286,429.785,176.866,18.245,152.519
C00629=1094.661,196.038,429.809,176.863,18.245,152.520
C00630=1094.656,195.788,429.832,176.860,18.245,152.520
C00631=1094.651,195.540,429.855,176.857,18.244,152.521
C00632=1094.645,195.291,429.878,176.853,18.244,152.521
C00633=1094.639,195.042,429.902,176.851,18.243,152.522
C00634=1094.634,194.793,429.925,176.847,18.243,152.522
C00635=1094.628,194.544,429.948,176.844,18.243,152.523
C00636=1094.622,194.295,429.971,176.841,18.242,152.523
C00637=1094.617,194.047,429.994,176.838,18.242,152.524
C00638=1094.611,193.798,430.018,176.835,18.241,152.524
C00639=1094.606,193.549,430.041,176.832,18.241,152.525
C00640=1094.600,193.300,430.064,176.829,18.240,152.525
C00641=1094.594,193.051,430.087,176.825,18.240,152.526
C00642=1094.589,192.802,430.111,176.822,18.239,152.526
C00643=1094.584,192.553,430.134,176.819,18.239,152.527
C00644=1094.577,192.278,430.159,176.816,18.238,152.527
C00645=1094.572,192.003,430.184,176.812,18.237,152.528
C00646=1094.565,191.729,430.210,176.809,18.237,152.528
C00647=1094.559,191.453,430.235,176.806,18.237,152.529
C00648=1094.553,191.204,430.258,176.803,18.236,152.529
C00649=1094.548,190.955,430.281,176.799,18.236,152.530
C00650=1094.543,190.706,430.305,176.796,18.235,152.530
C00651=1094.537,190.457,430.328,176.793,18.235,152.531
C00652=1094.531,190.208,430.351,176.790,18.234,152.531
C00653=1094.526,189.959,430.374,176.787,18.234,152.532
C00654=1094.520,189.710,430.397,176.784,18.233,152.532
C00655=1094.515,189.462,430.419,176.781,18.233,152.533
C00656=1094.510,189.213,430.443,176.778,18.232,152.533
C00657=1094.504,188.964,430.466,176.774,18.232,152.534
C00658=1094.498,188.715,430.489,176.771,18.231,152.534
C00659=1094.493,188.466,430.512,176.768,18.230,152.534
C00660=1094.487,188.217,430.535,176.765,18.230,152.535
C00661=1094.481,187.968,430.557,176.762,18.229,152.535
C00662=1094.476,187.720,430.580,176.759,18.229,152.536
C00663=1094.471,187.471,430.604,176.756,18.228,152.536
C00664=1094.465,187.222,430.627,176.753,18.228,152.537
C00665=1094.460,186.973,430.649,176.750,18.227,152.537
C00666=1094.454,186.724,430.672,176.747,18.227,152.538
C00667=1094.449,186.476,430.694,176.744,18.226,152.538
C00668=1094.443,186.227,430.717,176.740,18.226,152.539
C00669=1094.437,185.978,430.740,176.737,18.225,152.539
C00670=1094.432,185.729,430.763,176.734,18.224,152.539
C00671=1094.426,185.479,430.785,176.731,18.224,152.540
C00672=1094.421,185.231,430.808,176.728,18.223,152.540
C00673=1094.415,184.982,430.831,176.725,18.223,152.541
C00674=1094.410,184.733,430.854,176.722,18.222,152.541
C00675=1094.404,184.484,430.876,176.719,18.222,152.542
C00676=1094.399,184.235,430.899,176.716,18.221,152.542
C00677=1094.392,183.986,430.921,176.713,18.221,152.543
C00678=1094.386,183.737,430.944,176.710,18.220,152.543
C00679=1094.381,183.488,430.967,176.706,18.220,152.544
C00680=1094.375,183.239,430.990,176.703,18.219,152.544
C00681=1094.370,182.991,431.012,176.700,18.219,152.545
C00682=1094.364,182.742,431.034,176.697,18.218,152.545
C00683=1094.358,182.493,431.057,176.694,18.218,152.545
C00684=1094.352,182.244,431.080,176.692,18.218,152.546
C00685=1094.347,181.995,431.103,176.689,18.217,152.546
C00686=1094.341,181.746,431.124,176.685,18.217,152.547
C00687=1094.335,181.498,431.147,176.682,18.216,152.547
C00688=1094.330,181.248,431.169,176.679,18.216,152.548
C00689=1094.324,180.999,431.192,176.676,18.215,152.548
C00690=1094.318,180.751,431.214,176.673,18.215,152.549
C00691=1094.312,180.501,431.237,176.670,18.214,152.549
C00692=1094.307,180.252,431.259,176.667,18.213,152.550
C00693=1094.301,180.004,431.281,176.664,18.213,152.550
C00694=1094.295,179.755,431.304,176.661,18.213,152.551
C00695=1094.290,179.505,431.326,176.657,18.212,152.551
C00696=1094.283,179.257,431.348,176.654,18.212,152.552
C00697=1094.278,179.008,431.371,176.651,18.211,152.552
C00698=1094.273,178.759,431.393,176.648,18.211,152.553
C00699=1094.267,178.510,431.416,176.645,18.210,152.553
C00700=1094.261,178.261,431.438,176.642,18.209,152.553
C00701=1094.256,178.012,431.460,176.640,18.209,152.554
C00702=1094.250,177.763,431.482,176.637,18.209,152.554
C00703=1094.244,177.514,431.504,176.634,18.208,152.555
C00704=1094.239,177.265,431.527,176.631,18.208,152.555
C00705=1094.233,177.017,431.548,176.628,18.207,152.556
C00706=1094.227,176.768,431.571,176.625,18.206,152.556
C00707=1094.222,176.518,431.593,176.621,18.206,152.557
C00708=1094.215,176.243,431.618,176.618,18.205,152.557
C00709=1094.210,175.967,431.642,176.615,18.205,152.558
C00710=1094.203,175.692,431.667,176.611,18.204,152.558
C00711=1094.197,175.416,431.691,176.608,18.204,152.559
C00712=1094.191,175.167,431.714,176.605,18.203,152.559
C00713=1094.185,174.918,431.736,176.602,18.202,152.559
C00714=1094.181,174.669,431.758,176.599,18.202,152.560
C00715=1094.174,174.421,431.780,176.596,18.201,152.560
C00716=1094.169,174.172,431.802,176.593,18.201,152.561
C00717=1094.163,173.922,431.824,176.591,18.200,152.561
C00718=1094.157,173.674,431.847,176.588,18.200,152.562
C00719=1094.153,173.425,431.868,176.585,18.199,152.562
C00720=1094.146,173.176,431.890,176.581,18.199,152.562
C00721=1094.141,172.926,431.912,176.578,18.198,152.563
C00722=1094.135,172.678,431.934,176.575,18.197,152.563
C00723=1094.130,172.429,431.957,176.572,18.197,152.564
C00724=1094.124,172.179,431.978,176.569,18.196,152.564
C00725=1094.119,171.931,432.000,176.566,18.195,152.565
C00726=1094.112,171.682,432.022,176.563,18.195,152.565
C00727=1094.107,171.433,432.044,176.561,18.195,152.565
C00728=1094.102,171.184,432.066,176.558,18.194,152.566
C00729=1094.096,170.935,432.088,176.555,18.193,152.566
C00730=1094.091,170.686,432.110,176.552,18.193,152.567
C00731=1094.085,170.436,432.132,176.549,18.192,152.567
C00732=1094.080,170.188,432.153,176.546,18.191,152.567
C00733=1094.074,169.939,432.176,176.543,18.191,152.568
C00734=1094.069,169.690,432.198,176.540,18.190,152.568
C00735=1094.063,169.441,432.219,176.537,18.190,152.569
C00736=1094.058,169.192,432.241,176.534,18.189,152.569
C00737=1094.052,168.943,432.263,176.532,18.189,152.570
C00738=1094.047,168.694,432.285,176.529,18.188,152.570
C00739=1094.041,168.445,432.306,176.526,18.187,152.570
C00740=1094.036,168.196,432.328,176.523,18.187,152.571
C00741=1094.030,167.947,432.350,176.520,18.186,152.571
C00742=1094.025,167.698,432.372,176.517,18.185,152.572
C00743=1094.019,167.449,432.393,176.514,18.184,152.572
C00744=1094.014,167.200,432.415,176.511,18.184,152.572
C00745=1094.008,166.951,432.437,176.508,18.183,152.573
C00746=1094.003,166.702,432.459,176.506,18.183,152.573
C00747=1093.997,166.453,432.480,176.503,18.182,152.574
C00748=1093.992,166.204,432.502,176.500,18.181,152.574
C00749=1093.986,165.955,432.524,176.497,18.181,152.574
C00750=1093.980,165.706,432.545,176.494,18.180,152.575
C00751=1093.975,165.457,432.567,176.491,18.179,152.575
C00752=1093.969,165.208,432.589,176.488,18.179,152.576
C00753=1093.964,164.959,432.611,176.485,18.178,152.576
C00754=1093.958,164.710,432.632,176.482,18.178,152.577
C00755=1093.953,164.462,432.654,176.480,18.177,152.577
C00756=1093.947,164.212,432.675,176.477,18.176,152.577
C00757=1093.942,163.963,432.696,176.474,18.175,152.578
C00758=1093.936,163.714,432.718,176.471,18.174,152.578
C00759=1093.931,163.465,432.740,176.468,18.174,152.578
C00760=1093.926,163.216,432.761,176.465,18.173,152.579
C00761=1093.920,162.967,432.783,176.462,18.172,152.579
C00762=1093.915,162.718,432.804,176.460,18.172,152.580
C00763=1093.909,162.469,432.826,176.457,18.172,152.580
C00764=1093.904,162.220,432.847,176.454,18.171,152.580
C00765=1093.899,161.971,432.869,176.451,18.170,152.581
C00766=1093.893,161.721,432.890,176.448,18.169,152.581
C00767=1093.887,161.473,432.911,176.445,18.168,152.581
C00768=1093.881,161.224,432.933,176.442,18.168,152.582
C00769=1093.876,160.975,432.954,176.440,18.167,152.582
C00770=1093.871,160.726,432.975,176.437,18.167,152.583
C00771=1093.865,160.477,432.997,176.434,18.166,152.583
C00772=1093.858,160.201,433.021,176.431,18.165,152.584
C00773=1093.853,159.926,433.044,176.428,18.165,152.584
C00774=1093.846,159.649,433.067,176.424,18.164,152.585
C00775=1093.840,159.373,433.091,176.421,18.163,152.585
C00776=1093.834,159.125,433.113,176.418,18.162,152.585
C00777=1093.828,158.875,433.134,176.416,18.162,152.586
C00778=1093.823,158.626,433.155,176.413,18.161,152.586
C00779=1093.817,158.378,433.176,176.410,18.160,152.586
C00780=1093.811,158.128,433.197,176.407,18.160,152.587
C00781=1093.807,157.879,433.219,176.404,18.159,152.587
C00782=1093.801,157.629,433.240,176.401,18.158,152.588
C00783=1093.795,157.381,433.261,176.399,18.158,152.588
C00784=1093.790,157.132,433.282,176.396,18.157,152.588
C00785=1093.784,156.883,433.303,176.393,18.157,152.589
C00786=1093.778,156.634,433.325,176.390,18.156,152.589
C00787=1093.773,156.385,433.345,176.387,18.155,152.589
C00788=1093.767,156.136,433.367,176.384,18.154,152.590
C00789=1093.762,155.887,433.387,176.382,18.154,152.590
C00790=1093.756,155.638,433.409,176.379,18.153,152.591
C00791=1093.750,155.388,433.429,176.376,18.153,152.591
C00792=1093.745,155.140,433.451,176.373,18.151,152.591
C00793=1093.739,154.891,433.471,176.370,18.151,152.592
C00794=1093.733,154.641,433.493,176.367,18.150,152.592
C00795=1093.728,154.392,433.514,176.365,18.150,152.593
C00796=1093.722,154.144,433.535,176.362,18.149,152.593
C00797=1093.717,153.894,433.556,176.359,18.148,152.593
C00798=1093.711,153.645,433.577,176.356,18.147,152.594
C00799=1093.706,153.396,433.598,176.353,18.147,152.594
C00800=1093.700,153.147,433.619,176.351,18.146,152.594
C00801=1093.694,152.898,433.640,176.348,18.146,152.595
C00802=1093.689,152.649,433.660,176.345,18.145,152.595
C00803=1093.683,152.400,433.682,176.342,18.144,152.596
C00804=1093.678,152.151,433.702,176.339,18.143,152.596
C00805=1093.672,151.901,433.723,176.336,18.142,152.596
C00806=1093.667,151.653,433.744,176.334,18.142,152.597
C00807=1093.661,151.403,433.765,176.331,18.141,152.597
C00808=1093.655,151.155,433.786,176.328,18.140,152.597
C00809=1093.649,150.906,433.806,176.325,18.140,152.598
C00810=1093.644,150.657,433.827,176.323,18.139,152.598
C00811=1093.638,150.407,433.848,176.321,18.138,152.598
C00812=1093.633,150.158,433.869,176.318,18.138,152.599
C00813=1093.627,149.909,433.890,176.315,18.137,152.599
C00814=1093.622,149.660,433.910,176.312,18.136,152.600
C00815=1093.617,149.412,433.932,176.309,18.135,152.600
C00816=1093.610,149.162,433.952,176.307,18.135,152.600
C00817=1093.605,148.913,433.972,176.304,18.134,152.601
C00818=1093.600,148.664,433.993,176.301,18.133,152.601
C00819=1093.594,148.415,434.014,176.298,18.132,152.601
C00820=1093.588,148.166,434.035,176.295,18.131,152.602
C00821=1093.582,147.917,434.055,176.293,18.131,152.602
C00822=1093.577,147.668,434.076,176.290,18.130,152.602
C00823=1093.572,147.418,434.096,176.287,18.129,152.603
C00824=1093.565,147.169,434.118,176.284,18.129,152.603
C00825=1093.559,146.920,434.138,176.281,18.128,152.604
C00826=1093.554,146.671,434.158,176.279,18.127,152.604
C00827=1093.549,146.422,434.179,176.276,18.127,152.604
C00828=1093.543,146.173,434.199,176.273,18.126,152.605
C00829=1093.537,145.924,434.220,176.271,18.125,152.605
C00830=1093.532,145.674,434.240,176.269,18.125,152.605
C00831=1093.526,145.426,434.262,176.266,18.124,152.606
C00832=1093.520,145.177,434.282,176.263,18.123,152.606
C00833=1093.515,144.928,434.302,176.260,18.122,152.606
C00834=1093.510,144.679,434.323,176.257,18.121,152.607
C00835=1093.503,144.429,434.343,176.255,18.121,152.607
C00836=1093.497,144.154,434.366,176.252,18.120,152.607
C00837=1093.491,143.877,434.388,176.249,18.119,152.608
C00838=1093.486,143.601,434.411,176.245,18.118,152.608
C00839=1093.479,143.325,434.434,176.242,18.117,152.609
C00840=1093.473,143.076,434.454,176.240,18.117,152.609
C00841=1093.468,142.827,434.474,176.238,18.116,152.609
C00842=1093.463,142.577,434.495,176.235,18.115,152.610
C00843=1093.457,142.329,434.515,176.232,18.114,152.610
C00844=1093.451,142.079,434.536,176.229,18.113,152.610
C00845=1093.445,141.830,434.556,176.227,18.112,152.611
C00846=1093.440,141.581,434.576,176.224,18.112,152.611
C00847=1093.434,141.332,434.597,176.221,18.111,152.611
C00848=1093.428,141.083,434.617,176.218,18.110,152.612
C00849=1093.423,140.834,434.637,176.216,18.109,152.612
C00850=1093.418,140.585,434.658,176.213,18.109,152.612
C00851=1093.412,140.336,434.678,176.211,18.107,152.613
C00852=1093.407,140.087,434.698,176.208,18.107,152.613
C00853=1093.401,139.837,434.718,176.206,18.106,152.613
C00854=1093.396,139.588,434.738,176.203,18.105,152.614
C00855=1093.389,139.339,434.758,176.200,18.104,152.614
C00856=1093.384,139.090,434.779,176.197,18.104,152.614
C00857=1093.378,138.841,434.799,176.195,18.103,152.614
C00858=1093.372,138.592,434.819,176.192,18.102,152.615
C00859=1093.366,138.343,434.839,176.189,18.101,152.615
C00860=1093.362,138.093,434.859,176.186,18.100,152.616
C00861=1093.356,137.844,434.879,176.184,18.100,152.616
C00862=1093.350,137.595,434.900,176.181,18.099,152.616
C00863=1093.344,137.346,434.920,176.179,18.098,152.617
C00864=1093.339,137.097,434.940,176.176,18.097,152.617
C00865=1093.333,136.848,434.960,176.174,18.097,152.617
C00866=1093.327,136.599,434.979,176.171,18.095,152.617
C00867=1093.322,136.350,435.000,176.168,18.095,152.618
C00868=1093.316,136.101,435.020,176.165,18.094,152.618
C00869=1093.311,135.851,435.040,176.163,18.093,152.618
C00870=1093.305,135.602,435.060,176.160,18.092,152.619
C00871=1093.299,135.354,435.080,176.158,18.091,152.619
C00872=1093.294,135.104,435.100,176.155,18.090,152.619
C00873=1093.288,134.855,435.120,176.153,18.090,152.620
C00874=1093.283,134.606,435.140,176.150,18.089,152.620
C00875=1093.277,134.357,435.159,176.147,18.088,152.620
C00876=1093.271,134.108,435.179,176.144,18.087,152.621
C00877=1093.266,133.859,435.200,176.142,18.087,152.621
C00878=1093.260,133.609,435.219,176.139,18.086,152.621
C00879=1093.255,133.360,435.240,176.137,18.084,152.622
C00880=1093.249,133.111,435.260,176.134,18.084,152.622
C00881=1093.243,132.862,435.279,176.132,18.083,152.622
C00882=1093.238,132.613,435.299,176.129,18.082,152.622
C00883=1093.232,132.363,435.319,176.126,18.081,152.623
C00884=1093.226,132.114,435.339,176.124,18.081,152.623
C00885=1093.221,131.865,435.358,176.121,18.079,152.623
C00886=1093.216,131.616,435.378,176.118,18.079,152.624
C00887=1093.210,131.367,435.398,176.116,18.078,152.624
C00888=1093.204,131.118,435.418,176.114,18.077,152.624
C00889=1093.198,130.869,435.438,176.111,18.076,152.625
C00890=1093.192,130.619,435.457,176.108,18.075,152.625
C00891=1093.187,130.370,435.477,176.106,18.075,152.625
C00892=1093.181,130.121,435.497,176.103,18.074,152.626
C00893=1093.175,129.872,435.517,176.100,18.073,152.626
C00894=1093.170,129.623,435.536,176.097,18.072,152.626
C00895=1093.164,129.374,435.556,176.095,18.071,152.627
C00896=1093.158,129.124,435.575,176.093,18.070,152.627
C00897=1093.153,128.875,435.596,176.090,18.069,152.627
C00898=1093.147,128.626,435.615,176.088,18.069,152.627
C00899=1093.141,128.376,435.634,176.085,18.068,152.628
C00900=1093.134,128.101,435.656,176.082,18.067,152.628
C00901=1093.128,127.824,435.678,176.079,18.066,152.628
C00902=1093.122,127.548,435.699,176.077,18.065,152.629
C00903=1093.116,127.272,435.721,176.074,18.064,152.629
C00904=1093.110,127.022,435.740,176.071,18.063,152.629
C00905=1093.104,126.774,435.760,176.068,18.062,152.630
C00906=1093.099,126.524,435.780,176.066,18.061,152.630
C00907=1093.093,126.275,435.799,176.063,18.060,152.630
C00908=1093.087,126.026,435.819,176.060,18.059,152.631
C00909=1093.081,125.777,435.838,176.059,18.059,152.631
C00910=1093.076,125.527,435.858,176.056,18.057,152.631
C00911=1093.071,125.279,435.877,176.053,18.056,152.631
C00912=1093.065,125.029,435.897,176.051,18.056,152.632
C00913=1093.060,124.780,435.916,176.048,18.055,152.632
C00914=1093.054,124.531,435.936,176.045,18.054,152.632
C00915=1093.048,124.282,435.955,176.043,18.053,152.633
C00916=1093.042,124.032,435.974,176.041,18.052,152.633
C00917=1093.037,123.783,435.994,176.038,18.051,152.633
C00918=1093.031,123.535,436.013,176.035,18.050,152.633
C00919=1093.026,123.285,436.032,176.033,18.050,152.634
C00920=1093.020,123.036,436.052,176.030,18.048,152.634
C00921=1093.014,122.786,436.071,176.028,18.047,152.634
C00922=1093.008,122.538,436.091,176.026,18.047,152.634
C00923=1093.003,122.289,436.110,176.023,18.046,152.635
C00924=1092.997,122.039,436.129,176.020,18.044,152.635
C00925=1092.992,121.790,436.148,176.018,18.044,152.635
C00926=1092.986,121.540,436.168,176.016,18.043,152.636
C00927=1092.980,121.291,436.187,176.013,18.041,152.636
C00928=1092.975,121.043,436.206,176.010,18.040,152.636
C00929=1092.969,120.794,436.226,176.008,18.040,152.636
C00930=1092.964,120.544,436.245,176.006,18.039,152.637
C00931=1092.958,120.295,436.264,176.003,18.038,152.637
C00932=1092.953,120.046,436.283,176.001,18.037,152.637
C00933=1092.947,119.796,436.302,175.998,18.036,152.637
C00934=1092.941,119.547,436.321,175.995,18.035,152.638
C00935=1092.936,119.298,436.341,175.993,18.034,152.638
C00936=1092.931,119.049,436.360,175.991,18.033,152.638
C00937=1092.925,118.799,436.379,175.988,18.032,152.639
C00938=1092.919,118.550,436.398,175.986,18.031,152.639
C00939=1092.914,118.301,436.417,175.983,18.030,152.639
C00940=1092.908,118.052,436.437,175.981,18.029,152.639
C00941=1092.903,117.803,436.456,175.979,18.028,152.639
C00942=1092.897,117.554,436.475,175.976,18.027,152.640
C00943=1092.892,117.305,436.494,175.973,18.026,152.640
C00944=1092.886,117.055,436.514,175.971,18.025,152.640
C00945=1092.880,116.806,436.533,175.969,18.024,152.640
C00946=1092.876,116.557,436.551,175.966,18.023,152.641
C00947=1092.870,116.307,436.570,175.964,18.022,152.641
C00948=1092.864,116.058,436.589,175.961,18.021,152.641
C00949=1092.859,115.809,436.608,175.959,18.020,152.641
C00950=1092.853,115.560,436.628,175.957,18.019,152.642
C00951=1092.848,115.310,436.647,175.954,18.018,152.642
C00952=1092.843,115.061,436.666,175.951,18.016,152.642
C00953=1092.836,114.812,436.684,175.950,18.016,152.642
C00954=1092.831,114.563,436.704,175.947,18.015,152.643
C00955=1092.825,114.314,436.722,175.944,18.013,152.643
C00956=1092.820,114.065,436.742,175.942,18.013,152.643
C00957=1092.814,113.815,436.761,175.939,18.012,152.643
C00958=1092.808,113.566,436.779,175.937,18.010,152.644
C00959=1092.803,113.317,436.798,175.935,18.010,152.644
C00960=1092.797,113.067,436.817,175.932,18.009,152.644
C00961=1092.792,112.818,436.836,175.929,18.008,152.644
C00962=1092.786,112.570,436.854,175.928,18.006,152.645
C00963=1092.780,112.320,436.874,175.925,18.005,152.645
C00964=1092.774,112.044,436.894,175.922,18.004,152.645
C00965=1092.768,111.767,436.915,175.919,18.003,152.645
C00966=1092.761,111.491,436.936,175.917,18.002,152.646
C00967=1092.755,111.215,436.956,175.914,18.001,152.646
C00968=1092.750,110.965,436.976,175.912,18.000,152.646
C00969=1092.744,110.717,436.994,175.909,17.999,152.646
C00970=1092.738,110.467,437.013,175.907,17.998,152.647
C00971=1092.733,110.217,437.032,175.905,17.997,152.647
C00972=1092.727,109.969,437.050,175.902,17.996,152.647
C00973=1092.721,109.719,437.069,175.899,17.995,152.647
C00974=1092.716,109.470,437.088,175.898,17.994,152.648
C00975=1092.710,109.221,437.106,175.895,17.993,152.648
C00976=1092.704,108.971,437.125,175.893,17.992,152.648
C00977=1092.698,108.723,437.144,175.890,17.991,152.648
C00978=1092.693,108.473,437.162,175.887,17.990,152.649
C00979=1092.687,108.224,437.181,175.886,17.989,152.649
C00980=1092.682,107.975,437.200,175.883,17.987,152.649
C00981=1092.676,107.725,437.218,175.880,17.986,152.649
C00982=1092.670,107.477,437.236,175.878,17.986,152.649
C00983=1092.665,107.227,437.256,175.876,17.984,152.650
C00984=1092.659,106.977,437.274,175.873,17.983,152.650
C00985=1092.654,106.729,437.292,175.871,17.982,152.650
C00986=1092.648,106.479,437.311,175.869,17.981,152.650
C00987=1092.642,106.230,437.329,175.867,17.980,152.651
C00988=1092.637,105.981,437.349,175.864,17.979,152.651
C00989=1092.630,105.731,437.366,175.861,17.978,152.651
C00990=1092.625,105.482,437.385,175.860,17.977,152.651
C00991=1092.619,105.233,437.403,175.857,17.976,152.652
C00992=1092.614,104.984,437.422,175.854,17.974,152.652
C00993=1092.608,104.734,437.440,175.852,17.974,152.652
C00994=1092.603,104.485,437.459,175.850,17.972,152.652
C00995=1092.597,104.236,437.477,175.848,17.972,152.652
C00996=1092.592,103.987,437.496,175.845,17.970,152.653
C00997=1092.586,103.737,437.514,175.843,17.969,152.653
C00998=1092.581,103.488,437.533,175.841,17.968,152.653
C00999=1092.574,103.239,437.550,175.838,17.967,152.653
C01000=1092.569,102.990,437.569,175.835,17.966,152.653
C01001=1092.563,102.740,437.587,175.834,17.965,152.654
C01002=1092.558,102.492,437.606,175.831,17.963,152.654
C01003=1092.552,102.242,437.624,175.829,17.963,152.654
C01004=1092.547,101.992,437.642,175.827,17.961,152.654
C01005=1092.541,101.743,437.661,175.824,17.960,152.654
C01006=1092.536,101.494,437.679,175.822,17.959,152.655
C01007=1092.530,101.245,437.698,175.820,17.958,152.655
C01008=1092.525,100.995,437.716,175.817,17.957,152.655
C01009=1092.518,100.746,437.735,175.815,17.956,152.655
C01010=1092.513,100.497,437.752,175.812,17.954,152.655
C01011=1092.508,100.247,437.771,175.811,17.954,152.656
C01012=1092.502,99.999,437.789,175.808,17.953,152.656
C01013=1092.496,99.749,437.807,175.805,17.951,152.656
C01014=1092.491,99.500,437.825,175.803,17.950,152.656
C01015=1092.484,99.251,437.844,175.801,17.949,152.657
C01016=1092.479,99.002,437.861,175.799,17.948,152.657
C01017=1092.473,98.752,437.880,175.796,17.947,152.657
C01018=1092.468,98.503,437.898,175.794,17.946,152.657
C01019=1092.462,98.253,437.916,175.792,17.945,152.657
C01020=1092.457,98.004,437.934,175.789,17.944,152.658
C01021=1092.451,97.754,437.952,175.788,17.942,152.658
C01022=1092.445,97.506,437.970,175.785,17.941,152.658
C01023=1092.439,97.257,437.988,175.782,17.940,152.658
C01024=1092.434,97.007,438.006,175.780,17.939,152.658
C01025=1092.428,96.758,438.024,175.778,17.938,152.659
C01026=1092.422,96.509,438.043,175.776,17.937,152.659
C01027=1092.416,96.260,438.060,175.773,17.936,152.659
C01028=1092.410,95.983,438.081,175.771,17.934,152.659
C01029=1092.404,95.707,438.101,175.768,17.933,152.659
C01030=1092.398,95.431,438.121,175.765,17.932,152.660
C01031=1092.391,95.154,438.140,175.764,17.931,152.660
C01032=1092.386,94.905,438.159,175.761,17.929,152.660
C01033=1092.380,94.656,438.177,175.759,17.928,152.660
C01034=1092.375,94.407,438.194,175.757,17.927,152.660
C01035=1092.369,94.158,438.212,175.754,17.926,152.661
C01036=1092.364,93.907,438.230,175.752,17.925,152.661
C01037=1092.358,93.658,438.248,175.750,17.923,152.661
C01038=1092.352,93.409,438.266,175.747,17.922,152.661
C01039=1092.346,93.160,438.284,175.745,17.921,152.661
C01040=1092.341,92.911,438.302,175.743,17.919,152.661
C01041=1092.335,92.661,438.320,175.741,17.919,152.662
C01042=1092.330,92.412,438.338,175.739,17.917,152.662
C01043=1092.324,92.163,438.355,175.737,17.917,152.662
C01044=1092.318,91.913,438.373,175.734,17.915,152.662
C01045=1092.313,91.664,438.391,175.731,17.914,152.662
C01046=1092.308,91.415,438.409,175.730,17.913,152.662
C01047=1092.302,91.165,438.427,175.727,17.911,152.663
C01048=1092.296,90.916,438.445,175.725,17.910,152.663
C01049=1092.291,90.667,438.462,175.723,17.909,152.663
C01050=1092.285,90.417,438.480,175.721,17.908,152.663
C01051=1092.279,90.168,438.498,175.719,17.907,152.663
C01052=1092.274,89.919,438.515,175.716,17.905,152.664
C01053=1092.268,89.670,438.533,175.714,17.904,152.664
C01054=1092.262,89.421,438.551,175.711,17.903,152.664
C01055=1092.256,89.171,438.569,175.710,17.902,152.664
C01056=1092.250,88.922,438.586,175.707,17.901,152.664
C01057=1092.245,88.673,438.604,175.705,17.900,152.664
C01058=1092.239,88.423,438.622,175.703,17.899,152.665
C01059=1092.233,88.174,438.639,175.700,17.897,152.665
C01060=1092.228,87.925,438.657,175.699,17.896,152.665
C01061=1092.222,87.675,438.675,175.696,17.895,152.665
C01062=1092.216,87.426,438.692,175.694,17.894,152.665
C01063=1092.211,87.176,438.709,175.691,17.893,152.666
C01064=1092.205,86.927,438.727,175.690,17.891,152.666
C01065=1092.199,86.678,438.745,175.687,17.890,152.666
C01066=1092.194,86.429,438.762,175.685,17.889,152.666
C01067=1092.188,86.180,438.780,175.683,17.888,152.666
C01068=1092.182,85.930,438.798,175.681,17.886,152.666
C01069=1092.177,85.681,438.815,175.679,17.885,152.667
C01070=1092.171,85.431,438.832,175.676,17.884,152.667
C01071=1092.166,85.182,438.850,175.674,17.883,152.667
C01072=1092.160,84.932,438.868,175.672,17.881,152.667
C01073=1092.154,84.683,438.885,175.670,17.880,152.667
C01074=1092.149,84.434,438.903,175.668,17.879,152.667
C01075=1092.144,84.185,438.920,175.665,17.878,152.668
C01076=1092.137,83.935,438.937,175.663,17.876,152.668
C01077=1092.131,83.686,438.955,175.661,17.875,152.668
C01078=1092.126,83.437,438.972,175.659,17.874,152.668
C01079=1092.120,83.188,438.990,175.656,17.873,152.668
C01080=1092.114,82.938,439.007,175.655,17.871,152.668
C01081=1092.109,82.689,439.024,175.652,17.870,152.668
C01082=1092.103,82.440,439.042,175.650,17.869,152.669
C01083=1092.098,82.190,439.059,175.648,17.868,152.669
C01084=1092.093,81.941,439.076,175.646,17.866,152.669
C01085=1092.086,81.691,439.094,175.644,17.865,152.669
C01086=1092.081,81.442,439.112,175.641,17.864,152.669
C01087=1092.075,81.193,439.128,175.639,17.863,152.669
C01088=1092.069,80.944,439.146,175.637,17.861,152.669
C01089=1092.064,80.695,439.163,175.635,17.860,152.670
C01090=1092.058,80.444,439.181,175.633,17.859,152.670
C01091=1092.053,80.195,439.198,175.631,17.858,152.670
C01092=1092.047,79.919,439.217,175.628,17.856,152.670
C01093=1092.041,79.643,439.236,175.626,17.854,152.670
C01094=1092.034,79.367,439.256,175.624,17.853,152.670
C01095=1092.028,79.091,439.274,175.621,17.852,152.671
C01096=1092.022,78.842,439.292,175.619,17.850,152.671
C01097=1092.017,78.592,439.309,175.617,17.849,152.671
C01098=1092.011,78.343,439.326,175.615,17.848,152.671
C01099=1092.005,78.093,439.343,175.613,17.846,152.671
C01100=1092.000,77.844,439.361,175.611,17.845,152.671
C01101=1091.994,77.594,439.377,175.608,17.844,152.671
C01102=1091.988,77.345,439.394,175.607,17.843,152.671
C01103=1091.983,77.096,439.412,175.604,17.841,152.672
C01104=1091.977,76.847,439.429,175.602,17.841,152.672
C01105=1091.971,76.597,439.446,175.600,17.839,152.672
C01106=1091.965,76.348,439.463,175.598,17.838,152.672
C01107=1091.960,76.099,439.481,175.596,17.836,152.672
C01108=1091.954,75.849,439.497,175.594,17.835,152.672
C01109=1091.948,75.600,439.514,175.591,17.833,152.672
C01110=1091.943,75.351,439.531,175.590,17.833,152.673
C01111=1091.937,75.102,439.548,175.587,17.831,152.673
C01112=1091.931,74.851,439.565,175.585,17.830,152.673
C01113=1091.926,74.602,439.582,175.583,17.828,152.673
C01114=1091.920,74.353,439.599,175.581,17.827,152.673
C01115=1091.914,74.103,439.616,175.579,17.826,152.673
C01116=1091.909,73.854,439.634,175.576,17.824,152.673
C01117=1091.903,73.605,439.650,175.574,17.823,152.674
C01118=1091.897,73.356,439.668,175.572,17.822,152.674
C01119=1091.892,73.106,439.684,175.570,17.821,152.674
C01120=1091.886,72.857,439.701,175.568,17.819,152.674
C01121=1091.881,72.608,439.718,175.566,17.818,152.674
C01122=1091.875,72.359,439.734,175.564,17.816,152.674
C01123=1091.869,72.109,439.752,175.562,17.815,152.674
C01124=1091.863,71.859,439.769,175.560,17.814,152.674
C01125=1091.857,71.610,439.785,175.558,17.813,152.675
C01126=1091.852,71.361,439.803,175.556,17.811,152.675
C01127=1091.846,71.111,439.819,175.554,17.810,152.675
C01128=1091.841,70.862,439.836,175.551,17.809,152.675
C01129=1091.835,70.613,439.854,175.550,17.808,152.675
C01130=1091.829,70.363,439.870,175.547,17.806,152.675
C01131=1091.824,70.114,439.887,175.545,17.805,152.675
C01132=1091.818,69.864,439.903,175.543,17.803,152.675
C01133=1091.813,69.615,439.921,175.541,17.802,152.676
C01134=1091.807,69.366,439.937,175.539,17.800,152.676
C01135=1091.801,69.116,439.954,175.537,17.799,152.676
C01136=1091.796,68.867,439.970,175.535,17.798,152.676
C01137=1091.790,68.618,439.988,175.533,17.797,152.676
C01138=1091.784,68.369,440.004,175.531,17.795,152.676
C01139=1091.779,68.119,440.021,175.529,17.794,152.676
C01140=1091.773,67.870,440.037,175.526,17.792,152.676
C01141=1091.767,67.621,440.055,175.525,17.791,152.676
C01142=1091.761,67.371,440.071,175.522,17.789,152.677
C01143=1091.755,67.122,440.087,175.521,17.788,152.677
C01144=1091.750,66.872,440.104,175.518,17.787,152.677
C01145=1091.744,66.623,440.120,175.517,17.786,152.677
C01146=1091.739,66.374,440.138,175.514,17.784,152.677
C01147=1091.733,66.124,440.154,175.513,17.783,152.677
C01148=1091.728,65.875,440.171,175.510,17.781,152.677
C01149=1091.722,65.625,440.187,175.508,17.780,152.677
C01150=1091.716,65.376,440.203,175.506,17.779,152.677
C01151=1091.711,65.126,440.220,175.504,17.777,152.678
C01152=1091.705,64.877,440.236,175.502,17.776,152.678
C01153=1091.699,64.627,440.253,175.500,17.775,152.678
C01154=1091.693,64.379,440.270,175.498,17.773,152.678
C01155=1091.687,64.129,440.287,175.496,17.772,152.678
C01156=1091.680,63.852,440.304,175.494,17.770,152.678
C01157=1091.674,63.576,440.323,175.491,17.769,152.678
C01158=1091.668,63.300,440.341,175.489,17.768,152.678
C01159=1091.661,63.024,440.359,175.487,17.766,152.679
C01160=1091.656,62.774,440.376,175.485,17.765,152.679
C01161=1091.650,62.525,440.392,175.483,17.764,152.679
C01162=1091.644,62.276,440.409,175.481,17.763,152.679
C01163=1091.638,62.027,440.425,175.479,17.761,152.679
C01164=1091.633,61.777,440.442,175.477,17.760,152.679
C01165=1091.627,61.528,440.458,175.474,17.758,152.679
C01166=1091.621,61.278,440.475,175.473,17.757,152.679
C01167=1091.615,61.029,440.491,175.470,17.756,152.680
C01168=1091.609,60.780,440.507,175.469,17.754,152.680
C01169=1091.604,60.530,440.524,175.466,17.752,152.680
C01170=1091.598,60.281,440.540,175.465,17.751,152.680
C01171=1091.592,60.031,440.556,175.462,17.750,152.680
C01172=1091.586,59.781,440.572,175.461,17.748,152.680
C01173=1091.580,59.532,440.588,175.458,17.747,152.680
C01174=1091.574,59.283,440.605,175.457,17.746,152.680
C01175=1091.569,59.033,440.621,175.454,17.744,152.680
C01176=1091.563,58.784,440.638,175.452,17.743,152.680
C01177=1091.558,58.535,440.654,175.451,17.742,152.681
C01178=1091.552,58.286,440.670,175.448,17.740,152.681
C01179=1091.546,58.036,440.686,175.447,17.739,152.681
C01180=1091.540,57.787,440.702,175.444,17.738,152.681
C01181=1091.535,57.537,440.719,175.443,17.736,152.681
C01182=1091.529,57.287,440.735,175.440,17.735,152.681
C01183=1091.523,57.038,440.751,175.439,17.733,152.681
C01184=1091.517,56.789,440.767,175.436,17.732,152.681
C01185=1091.511,56.539,440.783,175.435,17.730,152.681
C01186=1091.505,56.290,440.800,175.432,17.729,152.681
C01187=1091.500,56.041,440.816,175.431,17.728,152.682
C01188=1091.494,55.791,440.831,175.429,17.727,152.682
C01189=1091.489,55.542,440.848,175.426,17.725,152.682
C01190=1091.483,55.292,440.864,175.425,17.723,152.682
C01191=1091.477,55.043,440.881,175.423,17.722,152.682
C01192=1091.471,54.794,440.897,175.421,17.721,152.682
C01193=1091.465,54.544,440.912,175.419,17.719,152.682
C01194=1091.460,54.295,440.928,175.417,17.718,152.682
C01195=1091.454,54.046,440.944,175.414,17.716,152.682
C01196=1091.448,53.796,440.961,175.413,17.715,152.682
C01197=1091.443,53.546,440.976,175.411,17.713,152.682
C01198=1091.437,53.297,440.993,175.409,17.712,152.682
C01199=1091.431,53.047,441.009,175.407,17.711,152.683
C01200=1091.426,52.798,441.025,175.405,17.709,152.683
C01201=1091.420,52.549,441.041,175.403,17.708,152.683
C01202=1091.414,52.299,441.057,175.401,17.706,152.683
C01203=1091.408,52.050,441.073,175.399,17.705,152.683
C01204=1091.403,51.800,441.089,175.397,17.703,152.683
C01205=1091.397,51.551,441.105,175.395,17.702,152.683
C01206=1091.392,51.302,441.121,175.393,17.700,152.683
C01207=1091.386,51.052,441.137,175.391,17.699,152.683
C01208=1091.380,50.803,441.153,175.390,17.698,152.683
C01209=1091.375,50.553,441.168,175.387,17.696,152.683
C01210=1091.369,50.304,441.184,175.386,17.695,152.683
C01211=1091.363,50.055,441.200,175.383,17.693,152.683
C01212=1091.357,49.805,441.216,175.382,17.692,152.684
C01213=1091.352,49.556,441.232,175.379,17.690,152.684
C01214=1091.346,49.306,441.247,175.378,17.689,152.684
C01215=1091.340,49.057,441.264,175.375,17.687,152.684
C01216=1091.334,48.807,441.280,175.374,17.686,152.684
C01217=1091.329,48.558,441.295,175.372,17.684,152.684
C01218=1091.323,48.309,441.311,175.370,17.683,152.684
C01219=1091.318,48.059,441.327,175.368,17.682,152.684
C01220=1091.312,47.782,441.345,175.366,17.679,152.684
C01221=1091.306,47.506,441.363,175.364,17.678,152.684
C01222=1091.299,47.229,441.380,175.362,17.677,152.684
C01223=1091.293,46.953,441.398,175.360,17.675,152.684
C01224=1091.288,46.704,441.413,175.358,17.674,152.684
C01225=1091.282,46.454,441.429,175.356,17.672,152.685
C01226=1091.276,46.205,441.445,175.354,17.670,152.684
C01227=1091.271,45.955,441.460,175.352,17.669,152.685
C01228=1091.265,45.706,441.477,175.350,17.668,152.685
C01229=1091.260,45.456,441.492,175.348,17.665,152.685
C01230=1091.254,45.207,441.507,175.346,17.664,152.685
C01231=1091.249,44.958,441.524,175.345,17.663,152.685
C01232=1091.243,44.708,441.539,175.343,17.661,152.685
C01233=1091.238,44.459,441.555,175.341,17.660,152.685
C01234=1091.232,44.209,441.571,175.339,17.658,152.685
C01235=1091.226,43.960,441.587,175.337,17.657,152.685
C01236=1091.220,43.711,441.601,175.335,17.655,152.685
C01237=1091.215,43.461,441.617,175.333,17.654,152.685
C01238=1091.209,43.211,441.633,175.332,17.652,152.685
C01239=1091.204,42.962,441.648,175.329,17.651,152.685
C01240=1091.198,42.713,441.665,175.328,17.649,152.685
C01241=1091.191,42.463,441.680,175.325,17.648,152.685
C01242=1091.186,42.214,441.695,175.324,17.646,152.686
C01243=1091.180,41.964,441.711,175.322,17.645,152.685
C01244=1091.175,41.714,441.727,175.320,17.643,152.686
C01245=1091.170,41.465,441.742,175.318,17.642,152.686
C01246=1091.163,41.216,441.757,175.316,17.640,152.686
C01247=1091.157,40.966,441.773,175.314,17.639,152.686
C01248=1091.152,40.717,441.788,175.313,17.638,152.686
C01249=1091.146,40.468,441.804,175.311,17.636,152.686
C01250=1091.140,40.218,441.819,175.309,17.635,152.686
C01251=1091.135,39.969,441.835,175.306,17.633,152.686
C01252=1091.129,39.719,441.850,175.305,17.631,152.686
C01253=1091.124,39.470,441.866,175.303,17.630,152.686
C01254=1091.117,39.220,441.881,175.301,17.628,152.686
C01255=1091.112,38.970,441.896,175.300,17.627,152.686
C01256=1091.107,38.721,441.912,175.297,17.625,152.686
C01257=1091.101,38.472,441.928,175.296,17.624,152.686
C01258=1091.095,38.223,441.942,175.293,17.622,152.686
C01259=1091.089,37.973,441.958,175.292,17.621,152.686
C01260=1091.084,37.723,441.974,175.290,17.619,152.686
C01261=1091.078,37.475,441.989,175.288,17.618,152.687
C01262=1091.072,37.225,442.004,175.286,17.616,152.687
C01263=1091.066,36.975,442.020,175.285,17.615,152.687
C01264=1091.061,36.726,442.034,175.282,17.613,152.687
C01265=1091.055,36.476,442.050,175.281,17.612,152.687
C01266=1091.049,36.227,442.065,175.278,17.610,152.687
C01267=1091.043,35.977,442.081,175.277,17.609,152.687
C01268=1091.037,35.728,442.096,175.275,17.608,152.687
C01269=1091.032,35.478,442.111,175.273,17.606,152.687
C01270=1091.026,35.229,442.127,175.272,17.604,152.687
C01271=1091.020,34.980,442.141,175.269,17.603,152.687
C01272=1091.015,34.730,442.157,175.268,17.602,152.687
C01273=1091.008,34.480,442.172,175.266,17.600,152.687
C01274=1091.003,34.231,442.187,175.264,17.598,152.687
C01275=1090.997,33.982,442.202,175.262,17.597,152.687
C01276=1090.991,33.732,442.218,175.261,17.596,152.687
C01277=1090.985,33.483,442.233,175.258,17.594,152.688
C01278=1090.980,33.233,442.248,175.257,17.592,152.687
C01279=1090.974,32.983,442.263,175.254,17.591,152.688
C01280=1090.968,32.734,442.278,175.253,17.589,152.688
C01281=1090.963,32.485,442.293,175.251,17.588,152.688
C01282=1090.957,32.235,442.308,175.249,17.586,152.688
C01283=1090.952,31.986,442.324,175.248,17.585,152.688
C01284=1090.944,31.709,442.340,175.245,17.583,152.688
C01285=1090.938,31.432,442.357,175.244,17.582,152.688
C01286=1090.932,31.156,442.373,175.241,17.579,152.688
C01287=1090.926,30.880,442.391,175.239,17.578,152.688
C01288=1090.920,30.631,442.405,175.238,17.576,152.688
C01289=1090.914,30.381,442.421,175.236,17.575,152.688
C01290=1090.909,30.132,442.435,175.234,17.574,152.688
C01291=1090.903,29.882,442.451,175.232,17.572,152.688
C01292=1090.897,29.633,442.465,175.231,17.571,152.688
C01293=1090.892,29.383,442.481,175.228,17.569,152.688
C01294=1090.886,29.134,442.495,175.227,17.568,152.688
C01295=1090.880,28.884,442.511,175.225,17.565,152.688
C01296=1090.875,28.635,442.525,175.223,17.564,152.688
C01297=1090.869,28.385,442.540,175.222,17.563,152.688
C01298=1090.863,28.136,442.555,175.219,17.561,152.688
C01299=1090.857,27.886,442.570,175.218,17.560,152.688
C01300=1090.852,27.637,442.585,175.216,17.558,152.688
C01301=1090.845,27.387,442.600,175.214,17.556,152.688
C01302=1090.840,27.138,442.615,175.212,17.555,152.689
C01303=1090.834,26.888,442.630,175.211,17.554,152.688
C01304=1090.828,26.639,442.645,175.208,17.552,152.689
C01305=1090.823,26.389,442.660,175.207,17.550,152.689
C01306=1090.817,26.140,442.674,175.205,17.549,152.689
C01307=1090.811,25.890,442.689,175.203,17.548,152.689
C01308=1090.806,25.641,442.704,175.202,17.546,152.689
C01309=1090.799,25.391,442.719,175.199,17.544,152.689
C01310=1090.793,25.142,442.734,175.198,17.543,152.689
C01311=1090.788,24.892,442.749,175.196,17.542,152.689
C01312=1090.782,24.643,442.763,175.194,17.540,152.689
C01313=1090.776,24.393,442.778,175.192,17.538,152.689
C01314=1090.770,24.144,442.793,175.191,17.537,152.689
C01315=1090.765,23.894,442.808,175.188,17.535,152.689
C01316=1090.759,23.644,442.822,175.187,17.534,152.689
C01317=1090.753,23.395,442.837,175.185,17.533,152.689
C01318=1090.748,23.146,442.852,175.183,17.530,152.689
C01319=1090.742,22.897,442.867,175.182,17.529,152.689
C01320=1090.736,22.646,442.881,175.180,17.528,152.689
C01321=1090.730,22.397,442.896,175.178,17.526,152.689
C01322=1090.725,22.148,442.911,175.176,17.524,152.689
C01323=1090.719,21.898,442.925,175.175,17.523,152.689
C01324=1090.713,21.649,442.940,175.173,17.521,152.689
C01325=1090.707,21.399,442.955,175.171,17.520,152.689
C01326=1090.702,21.150,442.970,175.170,17.519,152.689
C01327=1090.696,20.900,442.984,175.167,17.516,152.689
C01328=1090.690,20.651,442.999,175.166,17.515,152.690
C01329=1090.685,20.401,443.014,175.164,17.514,152.689
C01330=1090.679,20.151,443.028,175.162,17.512,152.690
C01331=1090.673,19.902,443.043,175.160,17.510,152.690
C01332=1090.667,19.653,443.057,175.159,17.509,152.690
C01333=1090.661,19.403,443.071,175.157,17.507,152.690
C01334=1090.655,19.154,443.086,175.155,17.506,152.690
C01335=1090.650,18.903,443.101,175.154,17.505,152.690
C01336=1090.644,18.654,443.115,175.151,17.503,152.690
C01337=1090.638,18.405,443.130,175.150,17.501,152.690
C01338=1090.632,18.155,443.144,175.148,17.500,152.690
C01339=1090.627,17.906,443.159,175.146,17.498,152.690
C01340=1090.621,17.657,443.173,175.145,17.496,152.690
C01341=1090.615,17.407,443.188,175.143,17.495,152.690
C01342=1090.610,17.157,443.202,175.141,17.493,152.690
C01343=1090.604,16.907,443.217,175.139,17.492,152.690
C01344=1090.598,16.659,443.232,175.138,17.491,152.690
C01345=1090.592,16.409,443.245,175.135,17.489,152.690
C01346=1090.586,16.159,443.260,175.134,17.487,152.690
C01347=1090.580,15.910,443.274,175.133,17.486,152.690
C01348=1090.575,15.635,443.290,175.130,17.484,152.690
C01349=1090.567,15.360,443.306,175.129,17.482,152.690
C01350=1090.562,15.085,443.322,175.126,17.481,152.690
C01351=1090.556,14.810,443.338,175.125,17.479,152.690
C01352=1090.549,14.560,443.353,175.123,17.477,152.690
C01353=1090.544,14.311,443.367,175.121,17.476,152.690
C01354=1090.538,14.062,443.381,175.120,17.474,152.690
C01355=1090.532,13.811,443.396,175.117,17.473,152.690
C01356=1090.527,13.562,443.409,175.116,17.471,152.690
C01357=1090.521,13.313,443.424,175.114,17.470,152.690
C01358=1090.514,13.063,443.438,175.112,17.468,152.690
C01359=1090.508,12.814,443.452,175.110,17.467,152.690
C01360=1090.503,12.564,443.466,175.109,17.465,152.690
C01361=1090.496,12.315,443.481,175.107,17.464,152.691
C01362=1090.491,12.065,443.495,175.105,17.462,152.691
C01363=1090.485,11.815,443.509,175.104,17.461,152.691
C01364=1090.479,11.566,443.524,175.102,17.459,152.691
C01365=1090.474,11.316,443.538,175.100,17.457,152.691
C01366=1090.468,11.067,443.552,175.098,17.456,152.691
C01367=1090.462,10.817,443.566,175.097,17.454,152.691
C01368=1090.456,10.567,443.580,175.095,17.453,152.691
C01369=1090.450,10.318,443.595,175.093,17.451,152.691
C01370=1090.444,10.069,443.608,175.092,17.450,152.691
C01371=1090.438,9.819,443.622,175.090,17.449,152.691
C01372=1090.432,9.570,443.637,175.088,17.447,152.691
C01373=1090.427,9.320,443.651,175.086,17.445,152.691
C01374=1090.421,9.070,443.665,175.085,17.444,152.691
C01375=1090.415,8.821,443.680,175.083,17.442,152.691
C01376=1090.410,8.572,443.693,175.081,17.440,152.691
C01377=1090.403,8.321,443.708,175.080,17.439,152.691
C01378=1090.398,8.072,443.722,175.078,17.438,152.691
C01379=1090.391,7.823,443.736,175.076,17.436,152.691
C01380=1090.386,7.574,443.749,175.074,17.434,152.691
C01381=1090.380,7.323,443.764,175.073,17.433,152.691
C01382=1090.374,7.074,443.778,175.071,17.431,152.691
C01383=1090.369,6.825,443.792,175.069,17.430,152.691
C01384=1090.363,6.575,443.806,175.068,17.429,152.691
C01385=1090.357,6.325,443.820,175.066,17.427,152.691
C01386=1090.351,6.076,443.834,175.064,17.425,152.691
C01387=1090.345,5.827,443.848,175.062,17.424,152.691
C01388=1090.340,5.577,443.862,175.061,17.422,152.691
C01389=1090.334,5.328,443.876,175.058,17.420,152.691
C01390=1090.328,5.077,443.890,175.057,17.419,152.691
C01391=1090.322,4.828,443.905,175.056,17.417,152.691
C01392=1090.316,4.579,443.918,175.054,17.416,152.691
C01393=1090.311,4.329,443.932,175.052,17.414,152.691
C01394=1090.305,4.080,443.946,175.050,17.413,152.691
C01395=1090.299,3.830,443.960,175.049,17.411,152.691
C01396=1090.294,3.580,443.974,175.047,17.409,152.691
C01397=1090.287,3.331,443.988,175.045,17.408,152.691
C01398=1090.282,3.082,444.001,175.044,17.407,152.691
C01399=1090.276,2.832,444.015,175.042,17.405,152.691
C01400=1090.271,2.583,444.029,175.040,17.403,152.691
C01401=1090.265,2.332,444.043,175.039,17.402,152.691
C01402=1090.258,2.083,444.057,175.037,17.400,152.691
C01403=1090.253,1.834,444.071,175.036,17.399,152.691
C01404=1090.247,1.584,444.084,175.033,17.397,152.691
C01405=1090.242,1.334,444.098,175.032,17.396,152.692
C01406=1090.236,1.085,444.112,175.030,17.394,152.692
C01407=1090.230,0.836,444.125,175.028,17.392,152.692
C01408=1090.224,0.587,444.140,175.027,17.391,152.692
C01409=1090.218,0.336,444.154,175.025,17.389,152.692
C01410=1090.213,0.087,444.168,175.024,17.388,152.691
C01411=1090.207,-0.163,444.181,175.021,17.386,152.692
C01412=1090.201,-0.436,444.196,175.020,17.384,152.692
C01413=1090.194,-0.709,444.211,175.018,17.382,152.692
C01414=1090.188,-0.982,444.227,175.016,17.381,152.692
C01415=1090.183,-1.255,444.242,175.015,17.380,152.692
C01416=1090.176,-1.504,444.255,175.013,17.377,152.692
C01417=1090.171,-1.754,444.269,175.011,17.376,152.692
C01418=1090.166,-2.003,444.283,175.010,17.375,152.692
C01419=1090.159,-2.253,444.296,175.007,17.373,152.692
C01420=1090.153,-2.503,444.310,175.006,17.371,152.692
C01421=1090.148,-2.752,444.324,175.004,17.370,152.692
C01422=1090.142,-3.002,444.338,175.003,17.368,152.692
C01423=1090.136,-3.251,444.351,175.001,17.366,152.692
C01424=1090.131,-3.501,444.365,174.999,17.365,152.692
C01425=1090.124,-3.750,444.378,174.998,17.363,152.692
C01426=1090.119,-4.000,444.392,174.996,17.362,152.692
C01427=1090.114,-4.250,444.405,174.994,17.360,152.692
C01428=1090.108,-4.499,444.419,174.993,17.359,152.692
C01429=1090.101,-4.749,444.433,174.991,17.358,152.692
C01430=1090.095,-4.999,444.446,174.990,17.356,152.692
C01431=1090.090,-5.248,444.460,174.987,17.354,152.692
C01432=1090.084,-5.498,444.473,174.986,17.353,152.692
C01433=1090.078,-5.747,444.487,174.984,17.351,152.692
C01434=1090.072,-5.996,444.500,174.983,17.350,152.692
C01435=1090.066,-6.246,444.514,174.981,17.348,152.692
C01436=1090.060,-6.496,444.527,174.979,17.347,152.692
C01437=1090.055,-6.745,444.541,174.978,17.345,152.692
C01438=1090.049,-6.995,444.554,174.976,17.344,152.692
C01439=1090.043,-7.244,444.568,174.975,17.342,152.692
C01440=1090.037,-7.494,444.581,174.972,17.340,152.692
C01441=1090.031,-7.744,444.595,174.971,17.339,152.692
C01442=1090.025,-7.994,444.608,174.969,17.338,152.692
C01443=1090.019,-8.243,444.621,174.968,17.336,152.692
C01444=1090.013,-8.493,444.635,174.966,17.334,152.692
C01445=1090.007,-8.742,444.648,174.964,17.333,152.692
C01446=1090.002,-8.992,444.661,174.963,17.331,152.692
C01447=1089.996,-9.241,444.675,174.961,17.330,152.692
C01448=1089.990,-9.491,444.688,174.960,17.328,152.692
C01449=1089.984,-9.740,444.702,174.957,17.327,152.692
C01450=1089.979,-9.990,444.715,174.956,17.325,152.692
C01451=1089.973,-10.240,444.728,174.955,17.324,152.692
C01452=1089.967,-10.489,444.742,174.953,17.323,152.692
C01453=1089.961,-10.738,444.755,174.951,17.320,152.692
C01454=1089.955,-10.988,444.768,174.950,17.319,152.692
C01455=1089.950,-11.238,444.782,174.948,17.318,152.692
C01456=1089.943,-11.487,444.795,174.947,17.316,152.692
C01457=1089.938,-11.737,444.808,174.944,17.314,152.692
C01458=1089.932,-11.987,444.821,174.943,17.313,152.692
C01459=1089.927,-12.236,444.835,174.941,17.311,152.692
C01460=1089.921,-12.486,444.848,174.940,17.310,152.692
C01461=1089.914,-12.735,444.861,174.938,17.309,152.692
C01462=1089.909,-12.985,444.875,174.936,17.306,152.692
C01463=1089.903,-13.235,444.887,174.935,17.305,152.693
C01464=1089.898,-13.484,444.901,174.933,17.304,152.692
C01465=1089.891,-13.734,444.915,174.932,17.302,152.692
C01466=1089.885,-13.983,444.927,174.930,17.301,152.692
C01467=1089.880,-14.233,444.941,174.928,17.299,152.692
C01468=1089.874,-14.482,444.954,174.927,17.297,152.692
C01469=1089.869,-14.732,444.967,174.925,17.296,152.693
C01470=1089.863,-14.981,444.980,174.924,17.295,152.692
C01471=1089.857,-15.231,444.993,174.921,17.292,152.692
C01472=1089.852,-15.481,445.007,174.920,17.291,152.693
C01473=1089.846,-15.730,445.019,174.918,17.290,152.693
C01474=1089.839,-15.980,445.033,174.917,17.289,152.693
C01475=1089.833,-16.229,445.046,174.915,17.287,152.693
C01476=1089.827,-16.502,445.060,174.913,17.285,152.693
C01477=1089.820,-16.773,445.074,174.912,17.284,152.693
C01478=1089.815,-17.044,445.089,174.910,17.282,152.693
C01479=1089.808,-17.315,445.103,174.908,17.280,152.693
C01480=1089.802,-17.565,445.115,174.906,17.279,152.693
C01481=1089.796,-17.814,445.129,174.905,17.277,152.693
C01482=1089.790,-18.064,445.142,174.903,17.276,152.693
C01483=1089.784,-18.314,445.155,174.901,17.274,152.693
C01484=1089.778,-18.563,445.168,174.900,17.272,152.693
C01485=1089.772,-18.813,445.181,174.898,17.271,152.693
C01486=1089.766,-19.063,445.193,174.897,17.270,152.693
C01487=1089.761,-19.312,445.207,174.895,17.269,152.693
C01488=1089.755,-19.562,445.220,174.893,17.266,152.693
C01489=1089.749,-19.811,445.233,174.892,17.265,152.693
C01490=1089.743,-20.061,445.245,174.890,17.264,152.693
C01491=1089.737,-20.310,445.258,174.889,17.262,152.693
C01492=1089.731,-20.560,445.271,174.887,17.261,152.693
C01493=1089.726,-20.809,445.285,174.885,17.259,152.693
C01494=1089.720,-21.059,445.297,174.884,17.257,152.693
C01495=1089.714,-21.309,445.310,174.882,17.256,152.693
C01496=1089.708,-21.558,445.323,174.881,17.255,152.693
C01497=1089.702,-21.808,445.336,174.879,17.254,152.693
C01498=1089.696,-22.057,445.349,174.878,17.252,152.693
C01499=1089.691,-22.307,445.362,174.875,17.250,152.693
C01500=1089.685,-22.557,445.374,174.874,17.249,152.693
C01501=1089.679,-22.806,445.388,174.872,17.247,152.693
C01502=1089.673,-23.056,445.400,174.871,17.246,152.693
C01503=1089.667,-23.305,445.414,174.869,17.244,152.693
C01504=1089.661,-23.555,445.426,174.867,17.242,152.693
C01505=1089.655,-23.805,445.439,174.866,17.241,152.693
C01506=1089.650,-24.054,445.452,174.864,17.240,152.693
C01507=1089.644,-24.304,445.465,174.863,17.238,152.693
C01508=1089.638,-24.554,445.477,174.861,17.237,152.693
C01509=1089.632,-24.803,445.491,174.860,17.235,152.693
C01510=1089.626,-25.053,445.503,174.857,17.234,152.693
C01511=1089.620,-25.303,445.516,174.856,17.232,152.693
C01512=1089.615,-25.552,445.528,174.855,17.230,152.693
C01513=1089.609,-25.801,445.541,174.853,17.229,152.693
C01514=1089.604,-26.051,445.554,174.852,17.228,152.693
C01515=1089.598,-26.301,445.567,174.850,17.227,152.693
C01516=1089.592,-26.551,445.579,174.848,17.224,152.693
C01517=1089.586,-26.800,445.592,174.846,17.223,152.693
C01518=1089.580,-27.049,445.605,174.845,17.222,152.694
C01519=1089.574,-27.299,445.617,174.843,17.220,152.693
C01520=1089.569,-27.549,445.630,174.842,17.219,152.694
C01521=1089.562,-27.799,445.643,174.840,17.217,152.694
C01522=1089.556,-28.048,445.656,174.838,17.216,152.694
C01523=1089.551,-28.298,445.668,174.837,17.214,152.694
C01524=1089.544,-28.547,445.680,174.835,17.213,152.694
C01525=1089.538,-28.796,445.693,174.834,17.211,152.694
C01526=1089.532,-29.046,445.706,174.832,17.210,152.694
C01527=1089.526,-29.296,445.718,174.831,17.209,152.694
C01528=1089.521,-29.546,445.731,174.829,17.207,152.694
C01529=1089.515,-29.795,445.743,174.827,17.205,152.694
C01530=1089.509,-30.045,445.756,174.826,17.204,152.694
C01531=1089.503,-30.294,445.769,174.824,17.203,152.694
C01532=1089.497,-30.544,445.781,174.823,17.201,152.694
C01533=1089.491,-30.794,445.794,174.821,17.200,152.694
C01534=1089.486,-31.043,445.806,174.820,17.198,152.694
C01535=1089.480,-31.293,445.819,174.818,17.197,152.694
C01536=1089.473,-31.543,445.831,174.816,17.195,152.694
C01537=1089.468,-31.793,445.843,174.814,17.194,152.694
C01538=1089.462,-32.041,445.856,174.813,17.193,152.694
C01539=1089.456,-32.291,445.869,174.811,17.191,152.694
C01540=1089.449,-32.562,445.883,174.810,17.190,152.694
C01541=1089.444,-32.833,445.896,174.808,17.188,152.694
C01542=1089.437,-33.103,445.909,174.806,17.186,152.694
C01543=1089.430,-33.374,445.923,174.805,17.185,152.694
C01544=1089.425,-33.623,445.935,174.803,17.183,152.694
C01545=1089.419,-33.873,445.947,174.801,17.182,152.694
C01546=1089.413,-34.123,445.960,174.799,17.180,152.694
C01547=1089.407,-34.373,445.972,174.798,17.179,152.694
C01548=1089.401,-34.622,445.984,174.796,17.177,152.694
C01549=1089.395,-34.872,445.997,174.795,17.176,152.694
C01550=1089.389,-35.122,446.009,174.793,17.175,152.694
C01551=1089.384,-35.371,446.021,174.792,17.173,152.694
C01552=1089.378,-35.621,446.034,174.790,17.172,152.694
C01553=1089.372,-35.870,446.046,174.788,17.170,152.694
C01554=1089.366,-36.120,446.059,174.787,17.169,152.694
C01555=1089.360,-36.369,446.071,174.785,17.167,152.694
C01556=1089.354,-36.619,446.083,174.784,17.166,152.694
C01557=1089.348,-36.869,446.096,174.782,17.164,152.695
C01558=1089.343,-37.118,446.108,174.781,17.163,152.694
C01559=1089.337,-37.368,446.120,174.779,17.162,152.695
C01560=1089.331,-37.618,446.132,174.778,17.160,152.695
C01561=1089.325,-37.867,446.145,174.775,17.158,152.695
C01562=1089.319,-38.117,446.157,174.774,17.157,152.695
C01563=1089.313,-38.367,446.170,174.772,17.156,152.695
C01564=1089.308,-38.616,446.182,174.771,17.154,152.695
C01565=1089.302,-38.865,446.194,174.769,17.153,152.695
C01566=1089.296,-39.115,446.206,174.768,17.151,152.695
C01567=1089.290,-39.364,446.219,174.766,17.150,152.695
C01568=1089.284,-39.615,446.230,174.765,17.149,152.695
C01569=1089.278,-39.864,446.242,174.763,17.148,152.695
C01570=1089.272,-40.114,446.255,174.761,17.146,152.695
C01571=1089.266,-40.363,446.267,174.760,17.144,152.695
C01572=1089.260,-40.613,446.279,174.758,17.143,152.695
C01573=1089.254,-40.863,446.292,174.757,17.142,152.695
C01574=1089.248,-41.112,446.303,174.755,17.140,152.695
C01575=1089.242,-41.362,446.316,174.754,17.139,152.695
C01576=1089.237,-41.612,446.328,174.752,17.137,152.695
C01577=1089.231,-41.861,446.339,174.751,17.136,152.695
C01578=1089.225,-42.111,446.352,174.749,17.135,152.695
C01579=1089.218,-42.361,446.364,174.748,17.134,152.695
C01580=1089.213,-42.610,446.376,174.746,17.132,152.695
C01581=1089.207,-42.860,446.388,174.744,17.130,152.695
C01582=1089.201,-43.110,446.400,174.742,17.129,152.695
C01583=1089.195,-43.359,446.412,174.741,17.128,152.695
C01584=1089.189,-43.609,446.424,174.739,17.126,152.695
C01585=1089.183,-43.858,446.436,174.738,17.125,152.695
C01586=1089.177,-44.108,446.449,174.736,17.123,152.695
C01587=1089.171,-44.358,446.460,174.735,17.122,152.696
C01588=1089.166,-44.607,446.472,174.733,17.121,152.696
C01589=1089.160,-44.857,446.485,174.732,17.120,152.696
C01590=1089.153,-45.106,446.497,174.730,17.118,152.696
C01591=1089.148,-45.356,446.508,174.729,17.117,152.696
C01592=1089.142,-45.606,446.520,174.726,17.115,152.696
C01593=1089.136,-45.856,446.533,174.725,17.114,152.696
C01594=1089.130,-46.105,446.543,174.723,17.112,152.696
C01595=1089.124,-46.355,446.556,174.722,17.111,152.696
C01596=1089.119,-46.604,446.568,174.720,17.110,152.696
C01597=1089.112,-46.854,446.580,174.719,17.108,152.696
C01598=1089.107,-47.104,446.592,174.717,17.107,152.696
C01599=1089.100,-47.353,446.604,174.716,17.105,152.696
C01600=1089.094,-47.603,446.616,174.714,17.104,152.696
C01601=1089.089,-47.853,446.627,174.713,17.103,152.696
C01602=1089.083,-48.103,446.640,174.711,17.102,152.696
C01603=1089.078,-48.352,446.652,174.710,17.100,152.696
C01604=1089.070,-48.623,446.664,174.708,17.098,152.696
C01605=1089.065,-48.894,446.677,174.706,17.097,152.696
C01606=1089.058,-49.165,446.690,174.705,17.096,152.696
C01607=1089.052,-49.436,446.703,174.703,17.094,152.696
C01608=1089.046,-49.685,446.715,174.702,17.093,152.696
C01609=1089.040,-49.936,446.726,174.700,17.092,152.696
C01610=1089.034,-50.184,446.738,174.698,17.090,152.696
C01611=1089.028,-50.434,446.751,174.696,17.089,152.697
C01612=1089.023,-50.684,446.761,174.695,17.087,152.696
C01613=1089.016,-50.933,446.773,174.693,17.086,152.697
C01614=1089.010,-51.184,446.785,174.692,17.085,152.697
C01615=1089.004,-51.433,446.797,174.690,17.083,152.697
C01616=1088.998,-51.682,446.809,174.689,17.082,152.697
C01617=1088.992,-51.933,446.821,174.687,17.081,152.697
C01618=1088.986,-52.182,446.832,174.686,17.079,152.697
C01619=1088.980,-52.432,446.843,174.684,17.078,152.697
C01620=1088.974,-52.681,446.855,174.682,17.077,152.697
C01621=1088.968,-52.931,446.867,174.681,17.076,152.697
C01622=1088.961,-53.181,446.879,174.679,17.074,152.697
C01623=1088.956,-53.430,446.890,174.678,17.073,152.697
C01624=1088.950,-53.680,446.902,174.676,17.072,152.697
C01625=1088.944,-53.929,446.914,174.675,17.071,152.697
C01626=1088.937,-54.179,446.925,174.673,17.070,152.697
C01627=1088.931,-54.428,446.937,174.672,17.068,152.697
C01628=1088.926,-54.679,446.949,174.670,17.067,152.697
C01629=1088.920,-54.927,446.960,174.668,17.066,152.698
C01630=1088.913,-55.178,446.971,174.667,17.064,152.697
C01631=1088.907,-55.428,446.983,174.665,17.063,152.698
C01632=1088.902,-55.677,446.995,174.664,17.062,152.698
C01633=1088.895,-55.927,447.006,174.662,17.060,152.698
C01634=1088.889,-56.176,447.018,174.661,17.059,152.698
C01635=1088.883,-56.426,447.029,174.658,17.058,152.698
C01636=1088.878,-56.676,447.041,174.657,17.056,152.698
C01637=1088.871,-56.926,447.052,174.655,17.055,152.698
C01638=1088.865,-57.175,447.064,174.654,17.054,152.698
C01639=1088.859,-57.425,447.075,174.652,17.052,152.698
C01640=1088.854,-57.675,447.087,174.651,17.051,152.698
C01641=1088.847,-57.924,447.099,174.649,17.050,152.698
C01642=1088.842,-58.174,447.109,174.648,17.048,152.698
C01643=1088.835,-58.423,447.121,174.646,17.047,152.698
C01644=1088.829,-58.673,447.132,174.644,17.046,152.698
C01645=1088.824,-58.923,447.144,174.643,17.045,152.698
C01646=1088.818,-59.172,447.156,174.641,17.043,152.699
C01647=1088.811,-59.422,447.167,174.640,17.042,152.699
C01648=1088.805,-59.672,447.178,174.638,17.041,152.699
C01649=1088.799,-59.921,447.190,174.637,17.040,152.699
C01650=1088.794,-60.171,447.201,174.635,17.039,152.699
C01651=1088.787,-60.421,447.213,174.634,17.037,152.699
C01652=1088.781,-60.670,447.224,174.632,17.036,152.699
C01653=1088.775,-60.920,447.235,174.631,17.035,152.699
C01654=1088.769,-61.170,447.246,174.629,17.034,152.699
C01655=1088.764,-61.419,447.258,174.628,17.032,152.699
C01656=1088.758,-61.669,447.270,174.626,17.031,152.699
C01657=1088.752,-61.919,447.281,174.624,17.030,152.699
C01658=1088.745,-62.168,447.292,174.623,17.028,152.699
C01659=1088.740,-62.418,447.303,174.621,17.027,152.699
C01660=1088.734,-62.668,447.315,174.620,17.026,152.699
C01661=1088.728,-62.917,447.327,174.618,17.025,152.700
C01662=1088.722,-63.167,447.338,174.617,17.023,152.699
C01663=1088.716,-63.417,447.349,174.615,17.022,152.700
C01664=1088.710,-63.666,447.360,174.613,17.021,152.700
C01665=1088.703,-63.916,447.372,174.612,17.020,152.700
C01666=1088.698,-64.165,447.383,174.610,17.018,152.700
C01667=1088.693,-64.415,447.394,174.609,17.017,152.700
C01668=1088.685,-64.688,447.406,174.607,17.016,152.700
C01669=1088.679,-64.960,447.419,174.606,17.015,152.700
C01670=1088.673,-65.232,447.431,174.604,17.014,152.700
C01671=1088.666,-65.504,447.443,174.603,17.012,152.700
C01672=1088.661,-65.754,447.454,174.601,17.011,152.700
C01673=1088.654,-66.004,447.466,174.600,17.010,152.700
C01674=1088.649,-66.254,447.477,174.598,17.009,152.700
C01675=1088.643,-66.503,447.487,174.596,17.008,152.700
C01676=1088.636,-66.753,447.499,174.595,17.006,152.700
C01677=1088.631,-67.002,447.510,174.593,17.005,152.700
C01678=1088.624,-67.252,447.522,174.592,17.004,152.701
C01679=1088.619,-67.502,447.532,174.590,17.002,152.701
C01680=1088.614,-67.752,447.544,174.589,17.001,152.701
C01681=1088.607,-68.002,447.555,174.587,17.000,152.701
C01682=1088.601,-68.251,447.566,174.585,16.999,152.701
C01683=1088.595,-68.500,447.578,174.584,16.997,152.701
C01684=1088.589,-68.750,447.589,174.582,16.996,152.701
C01685=1088.583,-69.000,447.600,174.581,16.995,152.701
C01686=1088.578,-69.249,447.611,174.579,16.994,152.701
C01687=1088.572,-69.499,447.621,174.578,16.992,152.701
C01688=1088.566,-69.749,447.633,174.576,16.991,152.701
C01689=1088.560,-69.998,447.644,174.575,16.990,152.701
C01690=1088.554,-70.248,447.654,174.573,16.989,152.701
C01691=1088.548,-70.498,447.666,174.572,16.987,152.701
C01692=1088.543,-70.748,447.677,174.570,16.986,152.701
C01693=1088.537,-70.997,447.688,174.568,16.985,152.702
C01694=1088.531,-71.248,447.699,174.567,16.984,152.702
C01695=1088.525,-71.497,447.710,174.565,16.982,152.702
C01696=1088.519,-71.746,447.722,174.564,16.981,152.702
C01697=1088.513,-71.995,447.733,174.562,16.980,152.702
C01698=1088.507,-72.246,447.744,174.560,16.979,152.702
C01699=1088.501,-72.495,447.755,174.559,16.978,152.702
C01700=1088.495,-72.745,447.766,174.557,16.976,152.702
C01701=1088.490,-72.994,447.777,174.556,16.975,152.702
C01702=1088.483,-73.244,447.788,174.555,16.975,152.702
C01703=1088.477,-73.494,447.799,174.553,16.974,152.702
C01704=1088.472,-73.744,447.809,174.552,16.972,152.702
C01705=1088.466,-73.993,447.820,174.550,16.971,152.702
C01706=1088.460,-74.244,447.831,174.549,16.970,152.703
C01707=1088.454,-74.493,447.842,174.547,16.969,152.703
C01708=1088.448,-74.743,447.853,174.545,16.968,152.703
C01709=1088.442,-74.993,447.864,174.544,16.967,152.703
C01710=1088.436,-75.242,447.875,174.542,16.966,152.703
C01711=1088.431,-75.492,447.886,174.541,16.964,152.703
C01712=1088.424,-75.742,447.896,174.539,16.963,152.703
C01713=1088.418,-75.991,447.907,174.537,16.962,152.703
C01714=1088.412,-76.241,447.918,174.536,16.961,152.703
C01715=1088.406,-76.490,447.929,174.534,16.960,152.703
C01716=1088.400,-76.740,447.940,174.533,16.958,152.703
C01717=1088.394,-76.990,447.951,174.532,16.958,152.704
C01718=1088.388,-77.239,447.961,174.530,16.957,152.704
C01719=1088.382,-77.488,447.972,174.528,16.956,152.704
C01720=1088.376,-77.739,447.983,174.527,16.954,152.704
C01721=1088.370,-77.989,447.994,174.525,16.953,152.704
C01722=1088.365,-78.238,448.005,174.524,16.952,152.704
C01723=1088.359,-78.488,448.015,174.522,16.951,152.704
C01724=1088.352,-78.738,448.026,174.521,16.950,152.704
C01725=1088.346,-78.987,448.037,174.519,16.949,152.704
C01726=1088.340,-79.237,448.048,174.517,16.947,152.704
C01727=1088.335,-79.487,448.058,174.516,16.946,152.704
C01728=1088.328,-79.737,448.069,174.514,16.945,152.705
C01729=1088.323,-79.986,448.080,174.513,16.945,152.705
C01730=1088.316,-80.236,448.090,174.512,16.944,152.705
C01731=1088.311,-80.485,448.101,174.510,16.943,152.705
C01732=1088.304,-80.760,448.113,174.508,16.941,152.705
C01733=1088.297,-81.035,448.124,174.507,16.940,152.705
C01734=1088.291,-81.309,448.136,174.504,16.939,152.705
C01735=1088.283,-81.583,448.148,174.503,16.938,152.705
C01736=1088.278,-81.833,448.158,174.501,16.936,152.705
C01737=1088.272,-82.082,448.169,174.500,16.936,152.706
C01738=1088.265,-82.332,448.180,174.499,16.935,152.706
C01739=1088.259,-82.582,448.190,174.497,16.934,152.706
C01740=1088.253,-82.831,448.201,174.495,16.933,152.706
C01741=1088.247,-83.081,448.211,174.494,16.932,152.706
C01742=1088.241,-83.331,448.222,174.492,16.930,152.706
C01743=1088.235,-83.581,448.233,174.490,16.929,152.706
C01744=1088.228,-83.830,448.243,174.489,16.928,152.706
C01745=1088.223,-84.080,448.253,174.487,16.927,152.706
C01746=1088.216,-84.330,448.264,174.486,16.927,152.706
C01747=1088.210,-84.579,448.275,174.485,16.925,152.707
C01748=1088.205,-84.830,448.285,174.483,16.924,152.707
C01749=1088.198,-85.079,448.295,174.481,16.923,152.707
C01750=1088.193,-85.328,448.306,174.480,16.922,152.707
C01751=1088.186,-85.579,448.316,174.478,16.921,152.707
C01752=1088.180,-85.828,448.327,174.476,16.920,152.707
C01753=1088.174,-86.078,448.338,174.475,16.919,152.707
C01754=1088.168,-86.327,448.348,174.474,16.918,152.707
C01755=1088.162,-86.577,448.358,174.472,16.917,152.707
C01756=1088.155,-86.827,448.369,174.471,16.916,152.707
C01757=1088.150,-87.077,448.379,174.469,16.915,152.708
C01758=1088.144,-87.326,448.390,174.467,16.914,152.708
C01759=1088.138,-87.576,448.400,174.466,16.913,152.708
C01760=1088.132,-87.826,448.411,174.464,16.912,152.708
C01761=1088.125,-88.076,448.421,174.462,16.911,152.708
C01762=1088.119,-88.325,448.432,174.461,16.911,152.708
C01763=1088.113,-88.575,448.442,174.460,16.910,152.708
C01764=1088.108,-88.824,448.453,174.458,16.908,152.708
C01765=1088.102,-89.075,448.463,174.457,16.907,152.709
C01766=1088.096,-89.324,448.473,174.455,16.906,152.709
C01767=1088.090,-89.573,448.484,174.453,16.905,152.709
C01768=1088.083,-89.824,448.494,174.452,16.904,152.709
C01769=1088.077,-90.073,448.505,174.451,16.903,152.709
C01770=1088.071,-90.323,448.514,174.449,16.902,152.709
C01771=1088.065,-90.572,448.525,174.448,16.901,152.709
C01772=1088.059,-90.822,448.535,174.446,16.901,152.709
C01773=1088.054,-91.072,448.546,174.444,16.900,152.710
C01774=1088.047,-91.321,448.556,174.442,16.898,152.710
C01775=1088.042,-91.571,448.566,174.442,16.898,152.710
C01776=1088.035,-91.821,448.577,174.440,16.897,152.710
C01777=1088.029,-92.071,448.587,174.438,16.896,152.710
C01778=1088.023,-92.321,448.598,174.437,16.895,152.710
C01779=1088.017,-92.570,448.607,174.435,16.894,152.710
C01780=1088.011,-92.820,448.618,174.433,16.892,152.710
C01781=1088.005,-93.070,448.628,174.431,16.892,152.711
C01782=1088.000,-93.319,448.639,174.431,16.891,152.711
C01783=1087.993,-93.569,448.648,174.429,16.890,152.711
C01784=1087.988,-93.818,448.659,174.427,16.889,152.711
C01785=1087.981,-94.068,448.669,174.426,16.888,152.711
C01786=1087.976,-94.318,448.679,174.424,16.887,152.711
C01787=1087.969,-94.568,448.689,174.422,16.886,152.711
C01788=1087.963,-94.818,448.700,174.422,16.885,152.711
C01789=1087.957,-95.067,448.710,174.420,16.885,152.712
C01790=1087.952,-95.318,448.720,174.418,16.884,152.712
C01791=1087.945,-95.567,448.730,174.416,16.882,152.712
C01792=1087.940,-95.817,448.740,174.415,16.881,152.712
C01793=1087.933,-96.066,448.751,174.414,16.881,152.712
C01794=1087.928,-96.316,448.761,174.412,16.880,152.712
C01795=1087.921,-96.565,448.771,174.410,16.879,152.712
C01796=1087.915,-96.842,448.782,174.409,16.878,152.712
C01797=1087.908,-97.119,448.793,174.407,16.877,152.713
C01798=1087.902,-97.396,448.805,174.406,16.876,152.713
C01799=1087.895,-97.673,448.816,174.404,16.875,152.713
C01800=1087.889,-97.922,448.826,174.402,16.874,152.713
C01801=1087.883,-98.172,448.836,174.400,16.873,152.713
C01802=1087.877,-98.422,448.846,174.399,16.872,152.713
C01803=1087.871,-98.671,448.856,174.398,16.871,152.713
C01804=1087.865,-98.921,448.866,174.396,16.871,152.714
C01805=1087.859,-99.170,448.876,174.394,16.870,152.714
C01806=1087.853,-99.420,448.886,174.393,16.869,152.714
C01807=1087.846,-99.671,448.896,174.391,16.868,152.714
C01808=1087.840,-99.920,448.906,174.390,16.867,152.714
C01809=1087.834,-100.170,448.916,174.388,16.866,152.714
C01810=1087.828,-100.420,448.926,174.387,16.865,152.714
C01811=1087.821,-100.669,448.936,174.385,16.864,152.714
C01812=1087.816,-100.919,448.946,174.383,16.864,152.715
C01813=1087.810,-101.169,448.956,174.382,16.863,152.715
C01814=1087.804,-101.418,448.966,174.381,16.862,152.715
C01815=1087.797,-101.668,448.976,174.379,16.861,152.715
C01816=1087.792,-101.918,448.986,174.377,16.860,152.715
C01817=1087.786,-102.168,448.996,174.376,16.860,152.715
C01818=1087.779,-102.417,449.006,174.374,16.859,152.716
